LIN {X 0,Y 573.137,Z 463.185,A -85,B 0,C 180,E1 -2255.983,E2 -2255.983} C_VEL
LIN {X 0,Y 573.164,Z 455.803,A -85,B 0,C 180,E1 -2256.86,E2 -2256.86} C_VEL
LIN {X 0,Y 573.212,Z 448.405,A -85,B 0,C 180,E1 -2257.574,E2 -2257.574} C_VEL
LIN {X 0,Y 573.278,Z 440.543,A -85,B 0,C 180,E1 -2258.193,E2 -2258.193} C_VEL
LIN {X 0,Y 573.324,Z 430.729,A -85,B 0,C 180,E1 -2258.814,E2 -2258.814} C_VEL
LIN {X 0,Y 573.388,Z 419.304,A -85,B 0,C 180,E1 -2259.346,E2 -2259.346} C_VEL
LIN {X 0,Y 573.473,Z 409.247,A -85,B 0,C 180,E1 -2259.679,E2 -2259.679} C_VEL
LIN {X 0,Y 573.529,Z 400.443,A -85,B 0,C 180,E1 -2259.878,E2 -2259.878} C_VEL
LIN {X 0,Y 573.641,Z 328.384,A -85,B 0,C 180,E1 -2260.797,E2 -2260.797} C_VEL
LIN {X 0,Y 573.174,Z 322.224,A -85,B 0,C 180,E1 -2260.899,E2 -2260.899} C_VEL
LIN {X 0,Y 573.324,Z 304.046,A -85,B 0,C 180,E1 -2263.649,E2 -2263.649} C_VEL
LIN {X 0,Y 573.504,Z 285.12,A -85,B 0,C 180,E1 -2266.544,E2 -2266.544} C_VEL
LIN {X 0,Y 573.63,Z 266.907,A -85,B 0,C 180,E1 -2269.371,E2 -2269.371} C_VEL
LIN {X 0,Y 573.846,Z 250.306,A -85,B 0,C 180,E1 -2271.934,E2 -2271.934} C_VEL
LIN {X 0,Y 573.51,Z 245.432,A -85,B 0,C 180,E1 -2272.706,E2 -2272.706} C_VEL
LIN {X 0,Y 573.237,Z 243.895,A -85,B 0,C 180,E1 -2272.98,E2 -2272.98} C_VEL
LIN {X 0,Y 573.248,Z 243.895,A -85,B 0,C 180,E1 -2275.41,E2 -2275.41} C_VEL
LIN {X 0,Y 573.231,Z 243.888,A -85,B 0,C 180,E1 -2278.564,E2 -2278.564} C_VEL
LIN {X 0,Y 573.223,Z 243.891,A -85,B 0,C 180,E1 -2280.993,E2 -2280.993} C_VEL
LIN {X 0,Y 573.262,Z 243.894,A -85,B 0,C 180,E1 -2283.524,E2 -2283.524} C_VEL
LIN {X 0,Y 573.239,Z 243.889,A -85,B 0,C 180,E1 -2286.049,E2 -2286.049} C_VEL
LIN {X 0,Y 573.236,Z 243.887,A -85,B 0,C 180,E1 -2288.701,E2 -2288.701} C_VEL
LIN {X 0,Y 573.251,Z 243.894,A -85,B 0,C 180,E1 -2291.595,E2 -2291.595} C_VEL
LIN {X 0,Y 573.233,Z 243.887,A -85,B 0,C 180,E1 -2294.333,E2 -2294.333} C_VEL
LIN {X 0,Y 573.236,Z 243.894,A -85,B 0,C 180,E1 -2297.358,E2 -2297.358} C_VEL
LIN {X 0,Y 573.242,Z 243.886,A -85,B 0,C 180,E1 -2300.392,E2 -2300.392} C_VEL
LIN {X 0,Y 573.251,Z 243.888,A -85,B 0,C 180,E1 -2303.077,E2 -2303.077} C_VEL
LIN {X 0,Y 573.263,Z 243.891,A -85,B 0,C 180,E1 -2305.671,E2 -2305.671} C_VEL
LIN {X 0,Y 573.238,Z 243.888,A -85,B 0,C 180,E1 -2308.184,E2 -2308.184} C_VEL
LIN {X 0,Y 573.261,Z 243.884,A -85,B 0,C 180,E1 -2310.634,E2 -2310.634} C_VEL
LIN {X 0,Y 573.265,Z 243.893,A -85,B 0,C 180,E1 -2313.5,E2 -2313.5} C_VEL
LIN {X 0,Y 573.228,Z 243.889,A -85,B 0,C 180,E1 -2316.134,E2 -2316.134} C_VEL
LIN {X 0,Y 573.247,Z 243.89,A -85,B 0,C 180,E1 -2319.173,E2 -2319.173} C_VEL
LIN {X 0,Y 573.225,Z 243.896,A -85,B 0,C 180,E1 -2321.411,E2 -2321.411} C_VEL
LIN {X 0,Y 573.247,Z 243.894,A -85,B 0,C 180,E1 -2323.621,E2 -2323.621} C_VEL
LIN {X 0,Y 573.267,Z 243.889,A -85,B 0,C 180,E1 -2325.806,E2 -2325.806} C_VEL
LIN {X 0,Y 573.256,Z 243.885,A -85,B 0,C 180,E1 -2328.744,E2 -2328.744} C_VEL
LIN {X 0,Y 573.3,Z 243.889,A -85,B 0,C 180,E1 -2331.54,E2 -2331.54} C_VEL
LIN {X 0,Y 573.284,Z 243.881,A -85,B 0,C 180,E1 -2334.371,E2 -2334.371} C_VEL
LIN {X 0,Y 573.302,Z 243.883,A -85,B 0,C 180,E1 -2337.892,E2 -2337.892} C_VEL
LIN {X 0,Y 573.329,Z 243.875,A -85,B 0,C 180,E1 -2340.702,E2 -2340.702} C_VEL
LIN {X 0,Y 573.232,Z 243.897,A -85,B 0,C 180,E1 -2343.514,E2 -2343.514} C_VEL
LIN {X 0,Y 573.283,Z 243.89,A -85,B 0,C 180,E1 -2345.628,E2 -2345.628} C_VEL
LIN {X 0,Y 573.284,Z 243.881,A -85,B 0,C 180,E1 -2348.459,E2 -2348.459} C_VEL
LIN {X 0,Y 573.263,Z 243.89,A -85,B 0,C 180,E1 -2351.311,E2 -2351.311} C_VEL
LIN {X 0,Y 573.264,Z 243.885,A -85,B 0,C 180,E1 -2354.192,E2 -2354.192} C_VEL
LIN {X 0,Y 573.251,Z 243.888,A -85,B 0,C 180,E1 -2357.111,E2 -2357.111} C_VEL
LIN {X 0,Y 573.248,Z 243.888,A -85,B 0,C 180,E1 -2360.076,E2 -2360.076} C_VEL
LIN {X 0,Y 573.229,Z 243.888,A -85,B 0,C 180,E1 -2362.337,E2 -2362.337} C_VEL
LIN {X 0,Y 573.242,Z 243.886,A -85,B 0,C 180,E1 -2364.398,E2 -2364.398} C_VEL
LIN {X 0,Y 572.617,Z 243.967,A -85,B 0,C 180,E1 -2364.985,E2 -2364.985} C_VEL
LIN {X 0,Y 569.778,Z 244.324,A -85,B 0,C 180,E1 -2365.936,E2 -2365.936} C_VEL
LIN {X 0,Y 567.349,Z 244.629,A -85,B 0,C 180,E1 -2366.702,E2 -2366.702} C_VEL
LIN {X 0,Y 566.297,Z 244.758,A -85,B 0,C 180,E1 -2367.293,E2 -2367.293} C_VEL
LIN {X 0,Y 566.208,Z 244.767,A -85,B 0,C 180,E1 -2367.494,E2 -2367.494} C_VEL
LIN {X 0,Y 566.179,Z 244.766,A -85,B 0,C 180,E1 -2370.592,E2 -2370.592} C_VEL
LIN {X 0,Y 566.22,Z 244.764,A -85,B 0,C 180,E1 -2373.101,E2 -2373.101} C_VEL
LIN {X 0,Y 566.204,Z 244.771,A -85,B 0,C 180,E1 -2375.688,E2 -2375.688} C_VEL
LIN {X 0,Y 566.206,Z 244.763,A -85,B 0,C 180,E1 -2378.559,E2 -2378.559} C_VEL
LIN {X 0,Y 566.202,Z 244.767,A -85,B 0,C 180,E1 -2381.136,E2 -2381.136} C_VEL
LIN {X 0,Y 566.19,Z 244.768,A -85,B 0,C 180,E1 -2384.035,E2 -2384.035} C_VEL
LIN {X 0,Y 566.2,Z 244.766,A -85,B 0,C 180,E1 -2387.082,E2 -2387.082} C_VEL
LIN {X 0,Y 566.217,Z 244.767,A -85,B 0,C 180,E1 -2389.803,E2 -2389.803} C_VEL
LIN {X 0,Y 566.189,Z 244.765,A -85,B 0,C 180,E1 -2392.599,E2 -2392.599} C_VEL
LIN {X 0,Y 566.203,Z 244.767,A -85,B 0,C 180,E1 -2395.182,E2 -2395.182} C_VEL
LIN {X 0,Y 566.227,Z 244.767,A -85,B 0,C 180,E1 -2397.744,E2 -2397.744} C_VEL
LIN {X 0,Y 566.194,Z 244.765,A -85,B 0,C 180,E1 -2400.328,E2 -2400.328} C_VEL
LIN {X 0,Y 566.21,Z 244.762,A -85,B 0,C 180,E1 -2402.661,E2 -2402.661} C_VEL
LIN {X 0,Y 566.226,Z 244.763,A -85,B 0,C 180,E1 -2405.039,E2 -2405.039} C_VEL
LIN {X 0,Y 566.192,Z 244.771,A -85,B 0,C 180,E1 -2407.369,E2 -2407.369} C_VEL
LIN {X 0,Y 566.211,Z 244.771,A -85,B 0,C 180,E1 -2409.663,E2 -2409.663} C_VEL
LIN {X 0,Y 566.191,Z 244.765,A -85,B 0,C 180,E1 -2412.668,E2 -2412.668} C_VEL
LIN {X 0,Y 566.224,Z 244.77,A -85,B 0,C 180,E1 -2415.627,E2 -2415.627} C_VEL
LIN {X 0,Y 566.267,Z 244.755,A -85,B 0,C 180,E1 -2418.654,E2 -2418.654} C_VEL
LIN {X 0,Y 566.224,Z 244.768,A -85,B 0,C 180,E1 -2421.434,E2 -2421.434} C_VEL
LIN {X 0,Y 566.243,Z 244.759,A -85,B 0,C 180,E1 -2424.301,E2 -2424.301} C_VEL
LIN {X 0,Y 566.268,Z 244.759,A -85,B 0,C 180,E1 -2427.154,E2 -2427.154} C_VEL
LIN {X 0,Y 566.273,Z 244.758,A -85,B 0,C 180,E1 -2430,E2 -2430} C_VEL
LIN {X 0,Y 566.261,Z 244.757,A -85,B 0,C 180,E1 -2432.845,E2 -2432.845} C_VEL
LIN {X 0,Y 566.244,Z 244.766,A -85,B 0,C 180,E1 -2435.698,E2 -2435.698} C_VEL
LIN {X 0,Y 566.195,Z 244.764,A -85,B 0,C 180,E1 -2438.566,E2 -2438.566} C_VEL
LIN {X 0,Y 566.232,Z 244.768,A -85,B 0,C 180,E1 -2441.454,E2 -2441.454} C_VEL
LIN {X 0,Y 566.208,Z 244.763,A -85,B 0,C 180,E1 -2444.5,E2 -2444.5} C_VEL
LIN {X 0,Y 566.186,Z 244.771,A -85,B 0,C 180,E1 -2447.332,E2 -2447.332} C_VEL
LIN {X 0,Y 566.199,Z 244.764,A -85,B 0,C 180,E1 -2450.337,E2 -2450.337} C_VEL
LIN {X 0,Y 566.157,Z 244.774,A -85,B 0,C 180,E1 -2453.281,E2 -2453.281} C_VEL
LIN {X 0,Y 566.193,Z 244.772,A -85,B 0,C 180,E1 -2455.749,E2 -2455.749} C_VEL
LIN {X 0,Y 566.191,Z 244.766,A -85,B 0,C 180,E1 -2458.202,E2 -2458.202} C_VEL
LIN {X 0,Y 566.178,Z 244.769,A -85,B 0,C 180,E1 -2461.076,E2 -2461.076} C_VEL
LIN {X 0,Y 566.19,Z 244.872,A -85,B 0,C 180,E1 -2463.205,E2 -2463.205} C_VEL
LIN {X 0,Y 566.004,Z 257.339,A -85,B 0,C 180,E1 -2466.189,E2 -2466.189} C_VEL
LIN {X 0,Y 565.966,Z 265.195,A -85,B 0,C 180,E1 -2468.054,E2 -2468.054} C_VEL
LIN {X 0,Y 566.66,Z 271.612,A -85,B 0,C 180,E1 -2468.154,E2 -2468.154} C_VEL
LIN {X 0,Y 566.526,Z 339.502,A -85,B 0,C 180,E1 -2469.027,E2 -2469.027} C_VEL
LIN {X 0,Y 566.417,Z 349.053,A -85,B 0,C 180,E1 -2469.239,E2 -2469.239} C_VEL
LIN {X 0,Y 566.403,Z 358.967,A -85,B 0,C 180,E1 -2469.57,E2 -2469.57} C_VEL
LIN {X 0,Y 566.3,Z 369.307,A -85,B 0,C 180,E1 -2470.041,E2 -2470.041} C_VEL
LIN {X 0,Y 566.244,Z 379.006,A -85,B 0,C 180,E1 -2470.637,E2 -2470.637} C_VEL
LIN {X 0,Y 566.155,Z 387.059,A -85,B 0,C 180,E1 -2471.258,E2 -2471.258} C_VEL
LIN {X 0,Y 566.113,Z 394.356,A -85,B 0,C 180,E1 -2471.947,E2 -2471.947} C_VEL
LIN {X 0,Y 566.027,Z 400.004,A -85,B 0,C 180,E1 -2472.584,E2 -2472.584} C_VEL
LIN {X 0,Y 565.976,Z 405.227,A -85,B 0,C 180,E1 -2473.286,E2 -2473.286} C_VEL
LIN {X 0,Y 565.962,Z 409.981,A -85,B 0,C 180,E1 -2474.057,E2 -2474.057} C_VEL
LIN {X 0,Y 565.9,Z 414.867,A -85,B 0,C 180,E1 -2475.062,E2 -2475.062} C_VEL
LIN {X 0,Y 565.896,Z 418.093,A -85,B 0,C 180,E1 -2475.936,E2 -2475.936} C_VEL
LIN {X 0,Y 565.857,Z 421.152,A -85,B 0,C 180,E1 -2477.119,E2 -2477.119} C_VEL
LIN {X 0,Y 565.849,Z 422.627,A -85,B 0,C 180,E1 -2478.176,E2 -2478.176} C_VEL
LIN {X 0,Y 565.824,Z 422.932,A -85,B 0,C 180,E1 -2479.258,E2 -2479.258} C_VEL
LIN {X 0,Y 565.858,Z 422.084,A -85,B 0,C 180,E1 -2480.356,E2 -2480.356} C_VEL
LIN {X 0,Y 565.899,Z 419.695,A -85,B 0,C 180,E1 -2481.615,E2 -2481.615} C_VEL
LIN {X 0,Y 565.921,Z 416.514,A -85,B 0,C 180,E1 -2482.634,E2 -2482.634} C_VEL
LIN {X 0,Y 565.937,Z 412.077,A -85,B 0,C 180,E1 -2483.642,E2 -2483.642} C_VEL
LIN {X 0,Y 565.987,Z 407.261,A -85,B 0,C 180,E1 -2484.494,E2 -2484.494} C_VEL
LIN {X 0,Y 566.037,Z 402.656,A -85,B 0,C 180,E1 -2485.171,E2 -2485.171} C_VEL
LIN {X 0,Y 566.085,Z 395.37,A -85,B 0,C 180,E1 -2486.037,E2 -2486.037} C_VEL
LIN {X 0,Y 566.135,Z 388.686,A -85,B 0,C 180,E1 -2486.689,E2 -2486.689} C_VEL
LIN {X 0,Y 566.24,Z 381.192,A -85,B 0,C 180,E1 -2487.293,E2 -2487.293} C_VEL
LIN {X 0,Y 566.33,Z 374.361,A -85,B 0,C 180,E1 -2487.751,E2 -2487.751} C_VEL
LIN {X 0,Y 566.344,Z 365.709,A -85,B 0,C 180,E1 -2488.223,E2 -2488.223} C_VEL
LIN {X 0,Y 566.379,Z 357.089,A -85,B 0,C 180,E1 -2488.591,E2 -2488.591} C_VEL
LIN {X 0,Y 566.474,Z 347.518,A -85,B 0,C 180,E1 -2488.891,E2 -2488.891} C_VEL
LIN {X 0,Y 566.541,Z 337.573,A -85,B 0,C 180,E1 -2489.096,E2 -2489.096} C_VEL
LIN {X 0,Y 566.548,Z 269.023,A -85,B 0,C 180,E1 -2489.97,E2 -2489.97} C_VEL
LIN {X 0,Y 565.997,Z 265.17,A -85,B 0,C 180,E1 -2490.041,E2 -2490.041} C_VEL
LIN {X 0,Y 566.136,Z 252.55,A -85,B 0,C 180,E1 -2493.042,E2 -2493.042} C_VEL
LIN {X 0,Y 566.185,Z 244.77,A -85,B 0,C 180,E1 -2494.949,E2 -2494.949} C_VEL
LIN {X 0,Y 566.169,Z 244.769,A -85,B 0,C 180,E1 -2497.369,E2 -2497.369} C_VEL
LIN {X 0,Y 566.209,Z 244.764,A -85,B 0,C 180,E1 -2499.664,E2 -2499.664} C_VEL
LIN {X 0,Y 566.194,Z 244.772,A -85,B 0,C 180,E1 -2502.669,E2 -2502.669} C_VEL
LIN {X 0,Y 566.222,Z 244.761,A -85,B 0,C 180,E1 -2505.627,E2 -2505.627} C_VEL
LIN {X 0,Y 566.264,Z 244.763,A -85,B 0,C 180,E1 -2508.655,E2 -2508.655} C_VEL
LIN {X 0,Y 566.239,Z 244.759,A -85,B 0,C 180,E1 -2511.435,E2 -2511.435} C_VEL
LIN {X 0,Y 566.251,Z 244.764,A -85,B 0,C 180,E1 -2514.302,E2 -2514.302} C_VEL
LIN {X 0,Y 566.271,Z 244.755,A -85,B 0,C 180,E1 -2517.867,E2 -2517.867} C_VEL
LIN {X 0,Y 566.298,Z 244.757,A -85,B 0,C 180,E1 -2520.712,E2 -2520.712} C_VEL
LIN {X 0,Y 566.27,Z 244.759,A -85,B 0,C 180,E1 -2522.846,E2 -2522.846} C_VEL
LIN {X 0,Y 566.252,Z 244.757,A -85,B 0,C 180,E1 -2525.699,E2 -2525.699} C_VEL
LIN {X 0,Y 566.239,Z 244.768,A -85,B 0,C 180,E1 -2528.566,E2 -2528.566} C_VEL
LIN {X 0,Y 566.232,Z 244.759,A -85,B 0,C 180,E1 -2531.455,E2 -2531.455} C_VEL
LIN {X 0,Y 566.225,Z 244.77,A -85,B 0,C 180,E1 -2534.507,E2 -2534.507} C_VEL
LIN {X 0,Y 566.196,Z 244.763,A -85,B 0,C 180,E1 -2537.332,E2 -2537.332} C_VEL
LIN {X 0,Y 566.212,Z 244.769,A -85,B 0,C 180,E1 -2540.338,E2 -2540.338} C_VEL
LIN {X 0,Y 566.182,Z 244.765,A -85,B 0,C 180,E1 -2543.405,E2 -2543.405} C_VEL
LIN {X 0,Y 566.219,Z 244.76,A -85,B 0,C 180,E1 -2545.749,E2 -2545.749} C_VEL
LIN {X 0,Y 566.201,Z 244.769,A -85,B 0,C 180,E1 -2548.204,E2 -2548.204} C_VEL
LIN {X 0,Y 566.181,Z 244.774,A -85,B 0,C 180,E1 -2550.593,E2 -2550.593} C_VEL
LIN {X 0,Y 566.223,Z 244.761,A -85,B 0,C 180,E1 -2553.102,E2 -2553.102} C_VEL
LIN {X 0,Y 566.206,Z 244.763,A -85,B 0,C 180,E1 -2555.689,E2 -2555.689} C_VEL
LIN {X 0,Y 566.209,Z 244.772,A -85,B 0,C 180,E1 -2558.56,E2 -2558.56} C_VEL
LIN {X 0,Y 566.203,Z 244.764,A -85,B 0,C 180,E1 -2561.137,E2 -2561.137} C_VEL
LIN {X 0,Y 566.192,Z 244.767,A -85,B 0,C 180,E1 -2564.037,E2 -2564.037} C_VEL
LIN {X 0,Y 566.197,Z 244.766,A -85,B 0,C 180,E1 -2567.084,E2 -2567.084} C_VEL
LIN {X 0,Y 566.203,Z 244.764,A -85,B 0,C 180,E1 -2569.802,E2 -2569.802} C_VEL
LIN {X 0,Y 566.195,Z 244.773,A -85,B 0,C 180,E1 -2572.6,E2 -2572.6} C_VEL
LIN {X 0,Y 566.204,Z 244.764,A -85,B 0,C 180,E1 -2575.183,E2 -2575.183} C_VEL
LIN {X 0,Y 566.227,Z 244.761,A -85,B 0,C 180,E1 -2577.744,E2 -2577.744} C_VEL
LIN {X 0,Y 566.2,Z 244.772,A -85,B 0,C 180,E1 -2580.329,E2 -2580.329} C_VEL
LIN {X 0,Y 566.195,Z 244.765,A -85,B 0,C 180,E1 -2583.344,E2 -2583.344} C_VEL
LIN {X 0,Y 566.198,Z 244.767,A -85,B 0,C 180,E1 -2585.82,E2 -2585.82} C_VEL
LIN {X 0,Y 566.223,Z 244.825,A -85,B 0,C 180,E1 -2587.049,E2 -2587.049} C_VEL
LIN {X 0,Y 566.789,Z 249.5,A -85,B 0,C 180,E1 -2587.779,E2 -2587.779} C_VEL
LIN {X 0,Y 566.638,Z 267.218,A -85,B 0,C 180,E1 -2590.498,E2 -2590.498} C_VEL
LIN {X 0,Y 566.491,Z 286.246,A -85,B 0,C 180,E1 -2593.421,E2 -2593.421} C_VEL
LIN {X 0,Y 566.283,Z 305.235,A -85,B 0,C 180,E1 -2596.361,E2 -2596.361} C_VEL
LIN {X 0,Y 566.128,Z 322.265,A -85,B 0,C 180,E1 -2598.97,E2 -2598.97} C_VEL
LIN {X 0,Y 566.696,Z 329.655,A -85,B 0,C 180,E1 -2599.085,E2 -2599.085} C_VEL
LIN {X 0,Y 566.59,Z 399.161,A -85,B 0,C 180,E1 -2599.977,E2 -2599.977} C_VEL
LIN {X 0,Y 566.469,Z 408.425,A -85,B 0,C 180,E1 -2600.178,E2 -2600.178} C_VEL
LIN {X 0,Y 566.425,Z 416.897,A -85,B 0,C 180,E1 -2600.448,E2 -2600.448} C_VEL
LIN {X 0,Y 566.358,Z 425.402,A -85,B 0,C 180,E1 -2600.807,E2 -2600.807} C_VEL
LIN {X 0,Y 566.318,Z 433.733,A -85,B 0,C 180,E1 -2601.256,E2 -2601.256} C_VEL
LIN {X 0,Y 566.212,Z 441.771,A -85,B 0,C 180,E1 -2601.794,E2 -2601.794} C_VEL
LIN {X 0,Y 566.12,Z 450.435,A -85,B 0,C 180,E1 -2602.51,E2 -2602.51} C_VEL
LIN {X 0,Y 566.088,Z 458.908,A -85,B 0,C 180,E1 -2603.402,E2 -2603.402} C_VEL
LIN {X 0,Y 566.057,Z 464.437,A -85,B 0,C 180,E1 -2604.121,E2 -2604.121} C_VEL
LIN {X 0,Y 565.906,Z 469.99,A -85,B 0,C 180,E1 -2605.013,E2 -2605.013} C_VEL
LIN {X 0,Y 565.944,Z 475.15,A -85,B 0,C 180,E1 -2606.084,E2 -2606.084} C_VEL
LIN {X 0,Y 565.88,Z 478.936,A -85,B 0,C 180,E1 -2607.153,E2 -2607.153} C_VEL
LIN {X 0,Y 565.841,Z 480.683,A -85,B 0,C 180,E1 -2607.865,E2 -2607.865} C_VEL
LIN {X 0,Y 565.844,Z 481.933,A -85,B 0,C 180,E1 -2608.577,E2 -2608.577} C_VEL
LIN {X 0,Y 565.837,Z 482.709,A -85,B 0,C 180,E1 -2609.289,E2 -2609.289} C_VEL
LIN {X 0,Y 565.836,Z 483,A -85,B 0,C 180,E1 -2610,E2 -2610} C_VEL
LIN {X 0,Y 565.837,Z 482.708,A -85,B 0,C 180,E1 -2610.712,E2 -2610.712} C_VEL
LIN {X 0,Y 565.844,Z 481.932,A -85,B 0,C 180,E1 -2611.424,E2 -2611.424} C_VEL
LIN {X 0,Y 565.841,Z 480.681,A -85,B 0,C 180,E1 -2612.136,E2 -2612.136} C_VEL
LIN {X 0,Y 565.912,Z 477.787,A -85,B 0,C 180,E1 -2613.204,E2 -2613.204} C_VEL
LIN {X 0,Y 565.944,Z 475.148,A -85,B 0,C 180,E1 -2613.916,E2 -2613.916} C_VEL
LIN {X 0,Y 565.906,Z 469.985,A -85,B 0,C 180,E1 -2614.987,E2 -2614.987} C_VEL
LIN {X 0,Y 566.082,Z 463.184,A -85,B 0,C 180,E1 -2616.058,E2 -2616.058} C_VEL
LIN {X 0,Y 566.092,Z 456.178,A -85,B 0,C 180,E1 -2616.906,E2 -2616.906} C_VEL
LIN {X 0,Y 566.146,Z 448.403,A -85,B 0,C 180,E1 -2617.669,E2 -2617.669} C_VEL
LIN {X 0,Y 566.258,Z 440.54,A -85,B 0,C 180,E1 -2618.296,E2 -2618.296} C_VEL
LIN {X 0,Y 566.327,Z 432.227,A -85,B 0,C 180,E1 -2618.834,E2 -2618.834} C_VEL
LIN {X 0,Y 566.374,Z 421.612,A -85,B 0,C 180,E1 -2619.373,E2 -2619.373} C_VEL
LIN {X 0,Y 566.473,Z 410.078,A -85,B 0,C 180,E1 -2619.777,E2 -2619.777} C_VEL
LIN {X 0,Y 566.559,Z 400.442,A -85,B 0,C 180,E1 -2620.001,E2 -2620.001} C_VEL
LIN {X 0,Y 566.686,Z 331.981,A -85,B 0,C 180,E1 -2620.885,E2 -2620.885} C_VEL
LIN {X 0,Y 566.411,Z 324.693,A -85,B 0,C 180,E1 -2620.983,E2 -2620.983} C_VEL
LIN {X 0,Y 566.137,Z 322.13,A -85,B 0,C 180,E1 -2621.051,E2 -2621.051} C_VEL
LIN {X 0,Y 566.319,Z 304.046,A -85,B 0,C 180,E1 -2623.821,E2 -2623.821} C_VEL
LIN {X 0,Y 566.512,Z 284.258,A -85,B 0,C 180,E1 -2626.889,E2 -2626.889} C_VEL
LIN {X 0,Y 566.634,Z 266.984,A -85,B 0,C 180,E1 -2629.565,E2 -2629.565} C_VEL
LIN {X 0,Y 566.902,Z 250.013,A -85,B 0,C 180,E1 -2632.217,E2 -2632.217} C_VEL
LIN {X 0,Y 566.191,Z 244.774,A -85,B 0,C 180,E1 -2633.099,E2 -2633.099} C_VEL
LIN {X 0,Y 566.207,Z 244.77,A -85,B 0,C 180,E1 -2635.749,E2 -2635.749} C_VEL
LIN {X 0,Y 566.203,Z 244.764,A -85,B 0,C 180,E1 -2638.202,E2 -2638.202} C_VEL
LIN {X 0,Y 566.189,Z 244.768,A -85,B 0,C 180,E1 -2641.076,E2 -2641.076} C_VEL
LIN {X 0,Y 566.211,Z 244.768,A -85,B 0,C 180,E1 -2643.734,E2 -2643.734} C_VEL
LIN {X 0,Y 566.207,Z 244.762,A -85,B 0,C 180,E1 -2646.569,E2 -2646.569} C_VEL
LIN {X 0,Y 566.212,Z 244.769,A -85,B 0,C 180,E1 -2649.685,E2 -2649.685} C_VEL
LIN {X 0,Y 566.211,Z 244.764,A -85,B 0,C 180,E1 -2652.087,E2 -2652.087} C_VEL
LIN {X 0,Y 566.171,Z 244.77,A -85,B 0,C 180,E1 -2655.035,E2 -2655.035} C_VEL
LIN {X 0,Y 566.209,Z 244.764,A -85,B 0,C 180,E1 -2658.136,E2 -2658.136} C_VEL
LIN {X 0,Y 566.216,Z 244.762,A -85,B 0,C 180,E1 -2660.726,E2 -2660.726} C_VEL
LIN {X 0,Y 566.203,Z 244.769,A -85,B 0,C 180,E1 -2663.784,E2 -2663.784} C_VEL
LIN {X 0,Y 566.207,Z 244.763,A -85,B 0,C 180,E1 -2666.265,E2 -2666.265} C_VEL
LIN {X 0,Y 566.186,Z 244.767,A -85,B 0,C 180,E1 -2668.923,E2 -2668.923} C_VEL
LIN {X 0,Y 566.224,Z 244.765,A -85,B 0,C 180,E1 -2671.858,E2 -2671.858} C_VEL
LIN {X 0,Y 566.221,Z 244.761,A -85,B 0,C 180,E1 -2674.251,E2 -2674.251} C_VEL
LIN {X 0,Y 566.186,Z 244.765,A -85,B 0,C 180,E1 -2676.713,E2 -2676.713} C_VEL
LIN {X 0,Y 566.21,Z 244.77,A -85,B 0,C 180,E1 -2679.662,E2 -2679.662} C_VEL
LIN {X 0,Y 566.194,Z 244.764,A -85,B 0,C 180,E1 -2682.668,E2 -2682.668} C_VEL
LIN {X 0,Y 566.228,Z 244.769,A -85,B 0,C 180,E1 -2685.626,E2 -2685.626} C_VEL
LIN {X 0,Y 566.228,Z 244.76,A -85,B 0,C 180,E1 -2688.674,E2 -2688.674} C_VEL
LIN {X 0,Y 566.241,Z 244.767,A -85,B 0,C 180,E1 -2691.434,E2 -2691.434} C_VEL
LIN {X 0,Y 566.253,Z 244.757,A -85,B 0,C 180,E1 -2694.301,E2 -2694.301} C_VEL
LIN {X 0,Y 566.274,Z 244.759,A -85,B 0,C 180,E1 -2697.866,E2 -2697.866} C_VEL
LIN {X 0,Y 566.299,Z 244.751,A -85,B 0,C 180,E1 -2700.71,E2 -2700.71} C_VEL
LIN {X 0,Y 566.271,Z 244.755,A -85,B 0,C 180,E1 -2702.845,E2 -2702.845} C_VEL
LIN {X 0,Y 566.251,Z 244.765,A -85,B 0,C 180,E1 -2705.698,E2 -2705.698} C_VEL
LIN {X 0,Y 566.228,Z 244.76,A -85,B 0,C 180,E1 -2708.565,E2 -2708.565} C_VEL
LIN {X 0,Y 566.233,Z 244.768,A -85,B 0,C 180,E1 -2711.454,E2 -2711.454} C_VEL
LIN {X 0,Y 566.225,Z 244.76,A -85,B 0,C 180,E1 -2714.506,E2 -2714.506} C_VEL
LIN {X 0,Y 566.196,Z 244.77,A -85,B 0,C 180,E1 -2717.331,E2 -2717.331} C_VEL
LIN {X 0,Y 566.211,Z 244.762,A -85,B 0,C 180,E1 -2720.336,E2 -2720.336} C_VEL
LIN {X 0,Y 566.18,Z 244.773,A -85,B 0,C 180,E1 -2723.403,E2 -2723.403} C_VEL
LIN {X 0,Y 566.217,Z 244.768,A -85,B 0,C 180,E1 -2725.748,E2 -2725.748} C_VEL
LIN {X 0,Y 566.208,Z 244.767,A -85,B 0,C 180,E1 -2727.494,E2 -2727.494} C_VEL
LIN {X 0,Y 565.528,Z 244.85,A -85,B 0,C 180,E1 -2728.087,E2 -2728.087} C_VEL
LIN {X 0,Y 562.657,Z 245.207,A -85,B 0,C 180,E1 -2729.051,E2 -2729.051} C_VEL
LIN {X 0,Y 560.243,Z 245.511,A -85,B 0,C 180,E1 -2729.826,E2 -2729.826} C_VEL
LIN {X 0,Y 559.215,Z 245.634,A -85,B 0,C 180,E1 -2730.425,E2 -2730.425} C_VEL
LIN {X 0,Y 559.136,Z 245.643,A -85,B 0,C 180,E1 -2730.628,E2 -2730.628} C_VEL
LIN {X 0,Y 559.169,Z 245.649,A -85,B 0,C 180,E1 -2733.573,E2 -2733.573} C_VEL
LIN {X 0,Y 559.16,Z 245.641,A -85,B 0,C 180,E1 -2736.448,E2 -2736.448} C_VEL
LIN {X 0,Y 559.168,Z 245.641,A -85,B 0,C 180,E1 -2738.933,E2 -2738.933} C_VEL
LIN {X 0,Y 559.182,Z 245.644,A -85,B 0,C 180,E1 -2741.767,E2 -2741.767} C_VEL
LIN {X 0,Y 559.13,Z 245.645,A -85,B 0,C 180,E1 -2744.739,E2 -2744.739} C_VEL
LIN {X 0,Y 559.158,Z 245.646,A -85,B 0,C 180,E1 -2747.257,E2 -2747.257} C_VEL
LIN {X 0,Y 559.176,Z 245.64,A -85,B 0,C 180,E1 -2750.135,E2 -2750.135} C_VEL
LIN {X 0,Y 559.134,Z 245.645,A -85,B 0,C 180,E1 -2752.892,E2 -2752.892} C_VEL
LIN {X 0,Y 559.157,Z 245.644,A -85,B 0,C 180,E1 -2756.05,E2 -2756.05} C_VEL
LIN {X 0,Y 559.154,Z 245.643,A -85,B 0,C 180,E1 -2758.981,E2 -2758.981} C_VEL
LIN {X 0,Y 559.183,Z 245.638,A -85,B 0,C 180,E1 -2762.288,E2 -2762.288} C_VEL
LIN {X 0,Y 559.169,Z 245.64,A -85,B 0,C 180,E1 -2764.813,E2 -2764.813} C_VEL
LIN {X 0,Y 559.153,Z 245.644,A -85,B 0,C 180,E1 -2767.068,E2 -2767.068} C_VEL
LIN {X 0,Y 559.177,Z 245.645,A -85,B 0,C 180,E1 -2769.396,E2 -2769.396} C_VEL
LIN {X 0,Y 559.139,Z 245.651,A -85,B 0,C 180,E1 -2771.686,E2 -2771.686} C_VEL
LIN {X 0,Y 559.161,Z 245.644,A -85,B 0,C 180,E1 -2773.948,E2 -2773.948} C_VEL
LIN {X 0,Y 559.163,Z 245.642,A -85,B 0,C 180,E1 -2776.184,E2 -2776.184} C_VEL
LIN {X 0,Y 559.201,Z 245.639,A -85,B 0,C 180,E1 -2779.134,E2 -2779.134} C_VEL
LIN {X 0,Y 559.196,Z 245.639,A -85,B 0,C 180,E1 -2782.053,E2 -2782.053} C_VEL
LIN {X 0,Y 559.246,Z 245.631,A -85,B 0,C 180,E1 -2784.953,E2 -2784.953} C_VEL
LIN {X 0,Y 559.236,Z 245.637,A -85,B 0,C 180,E1 -2787.839,E2 -2787.839} C_VEL
LIN {X 0,Y 559.26,Z 245.628,A -85,B 0,C 180,E1 -2790.72,E2 -2790.72} C_VEL
LIN {X 0,Y 559.228,Z 245.633,A -85,B 0,C 180,E1 -2792.881,E2 -2792.881} C_VEL
LIN {X 0,Y 559.211,Z 245.641,A -85,B 0,C 180,E1 -2795.77,E2 -2795.77} C_VEL
LIN {X 0,Y 559.16,Z 245.641,A -85,B 0,C 180,E1 -2798.674,E2 -2798.674} C_VEL
LIN {X 0,Y 559.195,Z 245.646,A -85,B 0,C 180,E1 -2801.6,E2 -2801.6} C_VEL
LIN {X 0,Y 559.169,Z 245.639,A -85,B 0,C 180,E1 -2804.587,E2 -2804.587} C_VEL
LIN {X 0,Y 559.145,Z 245.652,A -85,B 0,C 180,E1 -2807.557,E2 -2807.557} C_VEL
LIN {X 0,Y 559.157,Z 245.647,A -85,B 0,C 180,E1 -2809.837,E2 -2809.837} C_VEL
LIN {X 0,Y 559.128,Z 245.647,A -85,B 0,C 180,E1 -2812.153,E2 -2812.153} C_VEL
LIN {X 0,Y 559.136,Z 245.649,A -85,B 0,C 180,E1 -2815.299,E2 -2815.299} C_VEL
LIN {X 0,Y 559.13,Z 245.652,A -85,B 0,C 180,E1 -2817.714,E2 -2817.714} C_VEL
LIN {X 0,Y 559.138,Z 245.645,A -85,B 0,C 180,E1 -2820.183,E2 -2820.183} C_VEL
LIN {X 0,Y 559.146,Z 245.647,A -85,B 0,C 180,E1 -2823.144,E2 -2823.144} C_VEL
LIN {X 0,Y 559.081,Z 246.203,A -85,B 0,C 180,E1 -2823.364,E2 -2823.364} C_VEL
LIN {X 0,Y 558.961,Z 258.174,A -85,B 0,C 180,E1 -2826.223,E2 -2826.223} C_VEL
LIN {X 0,Y 558.906,Z 265.204,A -85,B 0,C 180,E1 -2827.916,E2 -2827.916} C_VEL
LIN {X 0,Y 559.692,Z 271.401,A -85,B 0,C 180,E1 -2828.015,E2 -2828.015} C_VEL
LIN {X 0,Y 559.549,Z 340.384,A -85,B 0,C 180,E1 -2828.916,E2 -2828.916} C_VEL
LIN {X 0,Y 559.438,Z 350.568,A -85,B 0,C 180,E1 -2829.157,E2 -2829.157} C_VEL
LIN {X 0,Y 559.348,Z 361.714,A -85,B 0,C 180,E1 -2829.558,E2 -2829.558} C_VEL
LIN {X 0,Y 559.265,Z 372.601,A -85,B 0,C 180,E1 -2830.122,E2 -2830.122} C_VEL
LIN {X 0,Y 559.194,Z 381.214,A -85,B 0,C 180,E1 -2830.694,E2 -2830.694} C_VEL
LIN {X 0,Y 559.093,Z 389.596,A -85,B 0,C 180,E1 -2831.385,E2 -2831.385} C_VEL
LIN {X 0,Y 558.975,Z 397.888,A -85,B 0,C 180,E1 -2832.236,E2 -2832.236} C_VEL
LIN {X 0,Y 558.912,Z 404.963,A -85,B 0,C 180,E1 -2833.172,E2 -2833.172} C_VEL
LIN {X 0,Y 558.867,Z 409.934,A -85,B 0,C 180,E1 -2833.985,E2 -2833.985} C_VEL
LIN {X 0,Y 558.846,Z 413.842,A -85,B 0,C 180,E1 -2834.768,E2 -2834.768} C_VEL
LIN {X 0,Y 558.81,Z 417.77,A -85,B 0,C 180,E1 -2835.795,E2 -2835.795} C_VEL
LIN {X 0,Y 558.799,Z 419.162,A -85,B 0,C 180,E1 -2836.234,E2 -2836.234} C_VEL
LIN {X 0,Y 558.753,Z 421.398,A -85,B 0,C 180,E1 -2837.219,E2 -2837.219} C_VEL
LIN {X 0,Y 558.753,Z 422.645,A -85,B 0,C 180,E1 -2838.194,E2 -2838.194} C_VEL
LIN {X 0,Y 558.741,Z 422.978,A -85,B 0,C 180,E1 -2839.152,E2 -2839.152} C_VEL
LIN {X 0,Y 558.752,Z 422.434,A -85,B 0,C 180,E1 -2840.107,E2 -2840.107} C_VEL
LIN {X 0,Y 558.758,Z 420.602,A -85,B 0,C 180,E1 -2841.243,E2 -2841.243} C_VEL
LIN {X 0,Y 558.818,Z 417.43,A -85,B 0,C 180,E1 -2842.401,E2 -2842.401} C_VEL
LIN {X 0,Y 558.845,Z 412.629,A -85,B 0,C 180,E1 -2843.595,E2 -2843.595} C_VEL
LIN {X 0,Y 558.912,Z 406.627,A -85,B 0,C 180,E1 -2844.661,E2 -2844.661} C_VEL
LIN {X 0,Y 558.95,Z 402.07,A -85,B 0,C 180,E1 -2845.324,E2 -2845.324} C_VEL
LIN {X 0,Y 559.014,Z 395.87,A -85,B 0,C 180,E1 -2846.072,E2 -2846.072} C_VEL
LIN {X 0,Y 559.091,Z 389.138,A -85,B 0,C 180,E1 -2846.745,E2 -2846.745} C_VEL
LIN {X 0,Y 559.214,Z 380.916,A -85,B 0,C 180,E1 -2847.418,E2 -2847.418} C_VEL
LIN {X 0,Y 559.321,Z 373.119,A -85,B 0,C 180,E1 -2847.936,E2 -2847.936} C_VEL
LIN {X 0,Y 559.34,Z 365.039,A -85,B 0,C 180,E1 -2848.372,E2 -2848.372} C_VEL
LIN {X 0,Y 559.429,Z 355.925,A -85,B 0,C 180,E1 -2848.754,E2 -2848.754} C_VEL
LIN {X 0,Y 559.49,Z 344.628,A -85,B 0,C 180,E1 -2849.094,E2 -2849.094} C_VEL
LIN {X 0,Y 559.544,Z 329.664,A -85,B 0,C 180,E1 -2849.333,E2 -2849.333} C_VEL
LIN {X 0,Y 559.654,Z 270.209,A -85,B 0,C 180,E1 -2850.091,E2 -2850.091} C_VEL
LIN {X 0,Y 558.935,Z 265.184,A -85,B 0,C 180,E1 -2850.178,E2 -2850.178} C_VEL
LIN {X 0,Y 559.056,Z 252.919,A -85,B 0,C 180,E1 -2853.093,E2 -2853.093} C_VEL
LIN {X 0,Y 559.096,Z 245.657,A -85,B 0,C 180,E1 -2854.699,E2 -2854.699} C_VEL
LIN {X 0,Y 559.111,Z 245.65,A -85,B 0,C 180,E1 -2857.067,E2 -2857.067} C_VEL
LIN {X 0,Y 559.175,Z 245.641,A -85,B 0,C 180,E1 -2859.396,E2 -2859.396} C_VEL
LIN {X 0,Y 559.145,Z 245.644,A -85,B 0,C 180,E1 -2861.687,E2 -2861.687} C_VEL
LIN {X 0,Y 559.161,Z 245.643,A -85,B 0,C 180,E1 -2863.949,E2 -2863.949} C_VEL
LIN {X 0,Y 559.163,Z 245.645,A -85,B 0,C 180,E1 -2866.185,E2 -2866.185} C_VEL
LIN {X 0,Y 559.2,Z 245.637,A -85,B 0,C 180,E1 -2869.134,E2 -2869.134} C_VEL
LIN {X 0,Y 559.2,Z 245.639,A -85,B 0,C 180,E1 -2872.054,E2 -2872.054} C_VEL
LIN {X 0,Y 559.251,Z 245.632,A -85,B 0,C 180,E1 -2874.954,E2 -2874.954} C_VEL
LIN {X 0,Y 559.243,Z 245.631,A -85,B 0,C 180,E1 -2877.84,E2 -2877.84} C_VEL
LIN {X 0,Y 559.268,Z 245.633,A -85,B 0,C 180,E1 -2880.721,E2 -2880.721} C_VEL
LIN {X 0,Y 559.236,Z 245.635,A -85,B 0,C 180,E1 -2882.882,E2 -2882.882} C_VEL
LIN {X 0,Y 559.221,Z 245.633,A -85,B 0,C 180,E1 -2885.771,E2 -2885.771} C_VEL
LIN {X 0,Y 559.194,Z 245.643,A -85,B 0,C 180,E1 -2888.675,E2 -2888.675} C_VEL
LIN {X 0,Y 559.196,Z 245.636,A -85,B 0,C 180,E1 -2891.601,E2 -2891.601} C_VEL
LIN {X 0,Y 559.19,Z 245.645,A -85,B 0,C 180,E1 -2894.596,E2 -2894.596} C_VEL
LIN {X 0,Y 559.155,Z 245.64,A -85,B 0,C 180,E1 -2897.557,E2 -2897.557} C_VEL
LIN {X 0,Y 559.167,Z 245.64,A -85,B 0,C 180,E1 -2899.838,E2 -2899.838} C_VEL
LIN {X 0,Y 559.135,Z 245.647,A -85,B 0,C 180,E1 -2902.153,E2 -2902.153} C_VEL
LIN {X 0,Y 559.172,Z 245.638,A -85,B 0,C 180,E1 -2905.188,E2 -2905.188} C_VEL
LIN {X 0,Y 559.188,Z 245.637,A -85,B 0,C 180,E1 -2907.712,E2 -2907.712} C_VEL
LIN {X 0,Y 559.159,Z 245.644,A -85,B 0,C 180,E1 -2910.183,E2 -2910.183} C_VEL
LIN {X 0,Y 559.169,Z 245.644,A -85,B 0,C 180,E1 -2912.715,E2 -2912.715} C_VEL
LIN {X 0,Y 559.151,Z 245.642,A -85,B 0,C 180,E1 -2915.323,E2 -2915.323} C_VEL
LIN {X 0,Y 559.129,Z 245.646,A -85,B 0,C 180,E1 -2918.018,E2 -2918.018} C_VEL
LIN {X 0,Y 559.17,Z 245.644,A -85,B 0,C 180,E1 -2920.811,E2 -2920.811} C_VEL
LIN {X 0,Y 559.136,Z 245.644,A -85,B 0,C 180,E1 -2923.735,E2 -2923.735} C_VEL
LIN {X 0,Y 559.141,Z 245.648,A -85,B 0,C 180,E1 -2926.804,E2 -2926.804} C_VEL
LIN {X 0,Y 559.155,Z 245.642,A -85,B 0,C 180,E1 -2929.189,E2 -2929.189} C_VEL
LIN {X 0,Y 559.129,Z 245.647,A -85,B 0,C 180,E1 -2931.983,E2 -2931.983} C_VEL
LIN {X 0,Y 559.143,Z 245.648,A -85,B 0,C 180,E1 -2934.786,E2 -2934.786} C_VEL
LIN {X 0,Y 559.171,Z 245.64,A -85,B 0,C 180,E1 -2937.362,E2 -2937.362} C_VEL
LIN {X 0,Y 559.145,Z 245.648,A -85,B 0,C 180,E1 -2940.144,E2 -2940.144} C_VEL
LIN {X 0,Y 559.163,Z 245.642,A -85,B 0,C 180,E1 -2943.175,E2 -2943.175} C_VEL
LIN {X 0,Y 559.156,Z 245.643,A -85,B 0,C 180,E1 -2945.496,E2 -2945.496} C_VEL
LIN {X 0,Y 559.202,Z 245.837,A -85,B 0,C 180,E1 -2946.998,E2 -2946.998} C_VEL
LIN {X 0,Y 559.777,Z 251.397,A -85,B 0,C 180,E1 -2947.874,E2 -2947.874} C_VEL
LIN {X 0,Y 559.602,Z 267.581,A -85,B 0,C 180,E1 -2950.377,E2 -2950.377} C_VEL
LIN {X 0,Y 559.477,Z 284.254,A -85,B 0,C 180,E1 -2952.952,E2 -2952.952} C_VEL
LIN {X 0,Y 559.318,Z 304.048,A -85,B 0,C 180,E1 -2956.003,E2 -2956.003} C_VEL
LIN {X 0,Y 559.09,Z 322.26,A -85,B 0,C 180,E1 -2958.828,E2 -2958.828} C_VEL
LIN {X 0,Y 559.72,Z 329.246,A -85,B 0,C 180,E1 -2958.942,E2 -2958.942} C_VEL
LIN {X 0,Y 559.611,Z 399.161,A -85,B 0,C 180,E1 -2959.851,E2 -2959.851} C_VEL
LIN {X 0,Y 559.494,Z 408.425,A -85,B 0,C 180,E1 -2960.054,E2 -2960.054} C_VEL
LIN {X 0,Y 559.441,Z 416.895,A -85,B 0,C 180,E1 -2960.327,E2 -2960.327} C_VEL
LIN {X 0,Y 559.363,Z 425.399,A -85,B 0,C 180,E1 -2960.691,E2 -2960.691} C_VEL
LIN {X 0,Y 559.308,Z 433.73,A -85,B 0,C 180,E1 -2961.146,E2 -2961.146} C_VEL
LIN {X 0,Y 559.198,Z 441.768,A -85,B 0,C 180,E1 -2961.69,E2 -2961.69} C_VEL
LIN {X 0,Y 559.094,Z 450.436,A -85,B 0,C 180,E1 -2962.416,E2 -2962.416} C_VEL
LIN {X 0,Y 559.034,Z 458.737,A -85,B 0,C 180,E1 -2963.297,E2 -2963.297} C_VEL
LIN {X 0,Y 559.004,Z 464.438,A -85,B 0,C 180,E1 -2964.047,E2 -2964.047} C_VEL
LIN {X 0,Y 558.822,Z 469.99,A -85,B 0,C 180,E1 -2964.95,E2 -2964.95} C_VEL
LIN {X 0,Y 558.859,Z 475.15,A -85,B 0,C 180,E1 -2966.034,E2 -2966.034} C_VEL
LIN {X 0,Y 558.803,Z 478.937,A -85,B 0,C 180,E1 -2967.117,E2 -2967.117} C_VEL
LIN {X 0,Y 558.747,Z 480.683,A -85,B 0,C 180,E1 -2967.838,E2 -2967.838} C_VEL
LIN {X 0,Y 558.744,Z 481.932,A -85,B 0,C 180,E1 -2968.559,E2 -2968.559} C_VEL
LIN {X 0,Y 558.737,Z 482.708,A -85,B 0,C 180,E1 -2969.279,E2 -2969.279} C_VEL
LIN {X 0,Y 558.737,Z 483,A -85,B 0,C 180,E1 -2970,E2 -2970} C_VEL
LIN {X 0,Y 558.737,Z 482.708,A -85,B 0,C 180,E1 -2970.721,E2 -2970.721} C_VEL
LIN {X 0,Y 558.744,Z 481.931,A -85,B 0,C 180,E1 -2971.442,E2 -2971.442} C_VEL
LIN {X 0,Y 558.747,Z 480.681,A -85,B 0,C 180,E1 -2972.163,E2 -2972.163} C_VEL
LIN {X 0,Y 558.836,Z 477.786,A -85,B 0,C 180,E1 -2973.244,E2 -2973.244} C_VEL
LIN {X 0,Y 558.859,Z 475.148,A -85,B 0,C 180,E1 -2973.966,E2 -2973.966} C_VEL
LIN {X 0,Y 558.822,Z 469.986,A -85,B 0,C 180,E1 -2975.051,E2 -2975.051} C_VEL
LIN {X 0,Y 559.018,Z 463.183,A -85,B 0,C 180,E1 -2976.135,E2 -2976.135} C_VEL
LIN {X 0,Y 559.036,Z 455.742,A -85,B 0,C 180,E1 -2977.04,E2 -2977.04} C_VEL
LIN {X 0,Y 559.119,Z 448.4,A -85,B 0,C 180,E1 -2977.766,E2 -2977.766} C_VEL
LIN {X 0,Y 559.227,Z 440.537,A -85,B 0,C 180,E1 -2978.401,E2 -2978.401} C_VEL
LIN {X 0,Y 559.292,Z 432.225,A -85,B 0,C 180,E1 -2978.946,E2 -2978.946} C_VEL
LIN {X 0,Y 559.385,Z 421.611,A -85,B 0,C 180,E1 -2979.491,E2 -2979.491} C_VEL
LIN {X 0,Y 559.5,Z 410.077,A -85,B 0,C 180,E1 -2979.9,E2 -2979.9} C_VEL
LIN {X 0,Y 559.578,Z 400.44,A -85,B 0,C 180,E1 -2980.127,E2 -2980.127} C_VEL
LIN {X 0,Y 559.745,Z 331.181,A -85,B 0,C 180,E1 -2981.032,E2 -2981.032} C_VEL
LIN {X 0,Y 559.357,Z 324.604,A -85,B 0,C 180,E1 -2981.124,E2 -2981.124} C_VEL
LIN {X 0,Y 559.091,Z 322.256,A -85,B 0,C 180,E1 -2981.172,E2 -2981.172} C_VEL
LIN {X 0,Y 559.336,Z 302.859,A -85,B 0,C 180,E1 -2984.183,E2 -2984.183} C_VEL
LIN {X 0,Y 559.478,Z 284.37,A -85,B 0,C 180,E1 -2987.053,E2 -2987.053} C_VEL
LIN {X 0,Y 559.643,Z 266.694,A -85,B 0,C 180,E1 -2989.82,E2 -2989.82} C_VEL
LIN {X 0,Y 559.923,Z 250.934,A -85,B 0,C 180,E1 -2992.314,E2 -2992.314} C_VEL
LIN {X 0,Y 559.139,Z 245.653,A -85,B 0,C 180,E1 -2993.221,E2 -2993.221} C_VEL
LIN {X 0,Y 559.172,Z 245.642,A -85,B 0,C 180,E1 -2996.097,E2 -2996.097} C_VEL
LIN {X 0,Y 559.138,Z 245.643,A -85,B 0,C 180,E1 -2998.531,E2 -2998.531} C_VEL
LIN {X 0,Y 559.144,Z 245.648,A -85,B 0,C 180,E1 -3001.273,E2 -3001.273} C_VEL
LIN {X 0,Y 559.165,Z 245.643,A -85,B 0,C 180,E1 -3003.949,E2 -3003.949} C_VEL
LIN {X 0,Y 559.142,Z 245.646,A -85,B 0,C 180,E1 -3007.108,E2 -3007.108} C_VEL
LIN {X 0,Y 559.158,Z 245.644,A -85,B 0,C 180,E1 -3009.941,E2 -3009.941} C_VEL
LIN {X 0,Y 559.159,Z 245.641,A -85,B 0,C 180,E1 -3012.743,E2 -3012.743} C_VEL
LIN {X 0,Y 559.15,Z 245.648,A -85,B 0,C 180,E1 -3015.76,E2 -3015.76} C_VEL
LIN {X 0,Y 559.183,Z 245.638,A -85,B 0,C 180,E1 -3018.231,E2 -3018.231} C_VEL
LIN {X 0,Y 559.173,Z 245.643,A -85,B 0,C 180,E1 -3021.191,E2 -3021.191} C_VEL
LIN {X 0,Y 559.157,Z 245.646,A -85,B 0,C 180,E1 -3023.79,E2 -3023.79} C_VEL
LIN {X 0,Y 559.158,Z 245.641,A -85,B 0,C 180,E1 -3026.424,E2 -3026.424} C_VEL
LIN {X 0,Y 559.151,Z 245.644,A -85,B 0,C 180,E1 -3028.98,E2 -3028.98} C_VEL
LIN {X 0,Y 559.166,Z 245.648,A -85,B 0,C 180,E1 -3031.618,E2 -3031.618} C_VEL
LIN {X 0,Y 559.195,Z 245.64,A -85,B 0,C 180,E1 -3033.903,E2 -3033.903} C_VEL
LIN {X 0,Y 559.152,Z 245.641,A -85,B 0,C 180,E1 -3036.567,E2 -3036.567} C_VEL
LIN {X 0,Y 559.175,Z 245.646,A -85,B 0,C 180,E1 -3039.395,E2 -3039.395} C_VEL
LIN {X 0,Y 559.143,Z 245.65,A -85,B 0,C 180,E1 -3041.685,E2 -3041.685} C_VEL
LIN {X 0,Y 559.162,Z 245.644,A -85,B 0,C 180,E1 -3043.947,E2 -3043.947} C_VEL
LIN {X 0,Y 559.166,Z 245.641,A -85,B 0,C 180,E1 -3046.183,E2 -3046.183} C_VEL
LIN {X 0,Y 559.19,Z 245.64,A -85,B 0,C 180,E1 -3049.133,E2 -3049.133} C_VEL
LIN {X 0,Y 559.202,Z 245.638,A -85,B 0,C 180,E1 -3052.053,E2 -3052.053} C_VEL
LIN {X 0,Y 559.25,Z 245.631,A -85,B 0,C 180,E1 -3054.953,E2 -3054.953} C_VEL
LIN {X 0,Y 559.245,Z 245.635,A -85,B 0,C 180,E1 -3057.839,E2 -3057.839} C_VEL
LIN {X 0,Y 559.269,Z 245.627,A -85,B 0,C 180,E1 -3060.719,E2 -3060.719} C_VEL
LIN {X 0,Y 559.237,Z 245.632,A -85,B 0,C 180,E1 -3062.881,E2 -3062.881} C_VEL
LIN {X 0,Y 559.221,Z 245.639,A -85,B 0,C 180,E1 -3065.77,E2 -3065.77} C_VEL
LIN {X 0,Y 559.186,Z 245.637,A -85,B 0,C 180,E1 -3068.674,E2 -3068.674} C_VEL
LIN {X 0,Y 559.197,Z 245.645,A -85,B 0,C 180,E1 -3071.6,E2 -3071.6} C_VEL
LIN {X 0,Y 559.191,Z 245.637,A -85,B 0,C 180,E1 -3074.595,E2 -3074.595} C_VEL
LIN {X 0,Y 559.156,Z 245.651,A -85,B 0,C 180,E1 -3077.556,E2 -3077.556} C_VEL
LIN {X 0,Y 559.166,Z 245.645,A -85,B 0,C 180,E1 -3079.837,E2 -3079.837} C_VEL
LIN {X 0,Y 559.134,Z 245.645,A -85,B 0,C 180,E1 -3082.152,E2 -3082.152} C_VEL
LIN {X 0,Y 559.17,Z 245.643,A -85,B 0,C 180,E1 -3085.187,E2 -3085.187} C_VEL
LIN {X 0,Y 559.185,Z 245.645,A -85,B 0,C 180,E1 -3087.711,E2 -3087.711} C_VEL
LIN {X 0,Y 559.136,Z 245.643,A -85,B 0,C 180,E1 -3090.628,E2 -3090.628} C_VEL
LIN {X 0,Y 558.478,Z 245.732,A -85,B 0,C 180,E1 -3091.229,E2 -3091.229} C_VEL
LIN {X 0,Y 555.618,Z 246.083,A -85,B 0,C 180,E1 -3092.205,E2 -3092.205} C_VEL
LIN {X 0,Y 553.207,Z 246.384,A -85,B 0,C 180,E1 -3092.991,E2 -3092.991} C_VEL
LIN {X 0,Y 552.188,Z 246.519,A -85,B 0,C 180,E1 -3093.598,E2 -3093.598} C_VEL
LIN {X 0,Y 552.115,Z 246.52,A -85,B 0,C 180,E1 -3093.803,E2 -3093.803} C_VEL
LIN {X 0,Y 552.102,Z 246.52,A -85,B 0,C 180,E1 -3096.746,E2 -3096.746} C_VEL
LIN {X 0,Y 552.14,Z 246.524,A -85,B 0,C 180,E1 -3099.525,E2 -3099.525} C_VEL
LIN {X 0,Y 552.121,Z 246.518,A -85,B 0,C 180,E1 -3102.425,E2 -3102.425} C_VEL
LIN {X 0,Y 552.09,Z 246.531,A -85,B 0,C 180,E1 -3105.563,E2 -3105.563} C_VEL
LIN {X 0,Y 552.131,Z 246.516,A -85,B 0,C 180,E1 -3108.676,E2 -3108.676} C_VEL
LIN {X 0,Y 552.11,Z 246.526,A -85,B 0,C 180,E1 -3111.411,E2 -3111.411} C_VEL
LIN {X 0,Y 552.091,Z 246.523,A -85,B 0,C 180,E1 -3114.157,E2 -3114.157} C_VEL
LIN {X 0,Y 552.114,Z 246.519,A -85,B 0,C 180,E1 -3116.815,E2 -3116.815} C_VEL
LIN {X 0,Y 552.098,Z 246.527,A -85,B 0,C 180,E1 -3119.391,E2 -3119.391} C_VEL
LIN {X 0,Y 552.117,Z 246.523,A -85,B 0,C 180,E1 -3121.903,E2 -3121.903} C_VEL
LIN {X 0,Y 552.146,Z 246.514,A -85,B 0,C 180,E1 -3124.649,E2 -3124.649} C_VEL
LIN {X 0,Y 552.105,Z 246.529,A -85,B 0,C 180,E1 -3127.55,E2 -3127.55} C_VEL
LIN {X 0,Y 552.148,Z 246.514,A -85,B 0,C 180,E1 -3130.674,E2 -3130.674} C_VEL
LIN {X 0,Y 552.111,Z 246.526,A -85,B 0,C 180,E1 -3133.737,E2 -3133.737} C_VEL
LIN {X 0,Y 552.127,Z 246.52,A -85,B 0,C 180,E1 -3136.004,E2 -3136.004} C_VEL
LIN {X 0,Y 552.169,Z 246.513,A -85,B 0,C 180,E1 -3138.994,E2 -3138.994} C_VEL
LIN {X 0,Y 552.15,Z 246.518,A -85,B 0,C 180,E1 -3141.951,E2 -3141.951} C_VEL
LIN {X 0,Y 552.22,Z 246.506,A -85,B 0,C 180,E1 -3144.889,E2 -3144.889} C_VEL
LIN {X 0,Y 552.209,Z 246.513,A -85,B 0,C 180,E1 -3147.812,E2 -3147.812} C_VEL
LIN {X 0,Y 552.231,Z 246.504,A -85,B 0,C 180,E1 -3150.729,E2 -3150.729} C_VEL
LIN {X 0,Y 552.195,Z 246.509,A -85,B 0,C 180,E1 -3152.918,E2 -3152.918} C_VEL
LIN {X 0,Y 552.179,Z 246.516,A -85,B 0,C 180,E1 -3155.844,E2 -3155.844} C_VEL
LIN {X 0,Y 552.135,Z 246.516,A -85,B 0,C 180,E1 -3158.786,E2 -3158.786} C_VEL
LIN {X 0,Y 552.152,Z 246.521,A -85,B 0,C 180,E1 -3161.75,E2 -3161.75} C_VEL
LIN {X 0,Y 552.118,Z 246.518,A -85,B 0,C 180,E1 -3164.748,E2 -3164.748} C_VEL
LIN {X 0,Y 552.095,Z 246.527,A -85,B 0,C 180,E1 -3167.788,E2 -3167.788} C_VEL
LIN {X 0,Y 552.117,Z 246.521,A -85,B 0,C 180,E1 -3170.101,E2 -3170.101} C_VEL
LIN {X 0,Y 552.079,Z 246.523,A -85,B 0,C 180,E1 -3172.451,E2 -3172.451} C_VEL
LIN {X 0,Y 552.103,Z 246.529,A -85,B 0,C 180,E1 -3175.645,E2 -3175.645} C_VEL
LIN {X 0,Y 552.078,Z 246.525,A -85,B 0,C 180,E1 -3178.099,E2 -3178.099} C_VEL
LIN {X 0,Y 552.089,Z 246.522,A -85,B 0,C 180,E1 -3180.609,E2 -3180.609} C_VEL
LIN {X 0,Y 552.049,Z 246.533,A -85,B 0,C 180,E1 -3183.257,E2 -3183.257} C_VEL
LIN {X 0,Y 551.911,Z 259.085,A -85,B 0,C 180,E1 -3186.255,E2 -3186.255} C_VEL
LIN {X 0,Y 551.847,Z 265.386,A -85,B 0,C 180,E1 -3187.767,E2 -3187.767} C_VEL
LIN {X 0,Y 552.766,Z 273.38,A -85,B 0,C 180,E1 -3187.899,E2 -3187.899} C_VEL
LIN {X 0,Y 552.568,Z 340.088,A -85,B 0,C 180,E1 -3188.781,E2 -3188.781} C_VEL
LIN {X 0,Y 552.427,Z 349.714,A -85,B 0,C 180,E1 -3189.005,E2 -3189.005} C_VEL
LIN {X 0,Y 552.367,Z 360.651,A -85,B 0,C 180,E1 -3189.39,E2 -3189.39} C_VEL
LIN {X 0,Y 552.258,Z 370.394,A -85,B 0,C 180,E1 -3189.87,E2 -3189.87} C_VEL
LIN {X 0,Y 552.16,Z 379.724,A -85,B 0,C 180,E1 -3190.475,E2 -3190.475} C_VEL
LIN {X 0,Y 552.118,Z 385.958,A -85,B 0,C 180,E1 -3190.96,E2 -3190.96} C_VEL
LIN {X 0,Y 551.979,Z 393.773,A -85,B 0,C 180,E1 -3191.701,E2 -3191.701} C_VEL
LIN {X 0,Y 551.895,Z 400.22,A -85,B 0,C 180,E1 -3192.446,E2 -3192.446} C_VEL
LIN {X 0,Y 551.836,Z 405.61,A -85,B 0,C 180,E1 -3193.198,E2 -3193.198} C_VEL
LIN {X 0,Y 551.785,Z 410.137,A -85,B 0,C 180,E1 -3193.959,E2 -3193.959} C_VEL
LIN {X 0,Y 551.771,Z 413.893,A -85,B 0,C 180,E1 -3194.725,E2 -3194.725} C_VEL
LIN {X 0,Y 551.72,Z 417.052,A -85,B 0,C 180,E1 -3195.526,E2 -3195.526} C_VEL
LIN {X 0,Y 551.698,Z 420.027,A -85,B 0,C 180,E1 -3196.56,E2 -3196.56} C_VEL
LIN {X 0,Y 551.647,Z 421.999,A -85,B 0,C 180,E1 -3197.638,E2 -3197.638} C_VEL
LIN {X 0,Y 551.655,Z 422.889,A -85,B 0,C 180,E1 -3198.732,E2 -3198.732} C_VEL
LIN {X 0,Y 551.636,Z 422.672,A -85,B 0,C 180,E1 -3199.854,E2 -3199.854} C_VEL
LIN {X 0,Y 551.657,Z 421.206,A -85,B 0,C 180,E1 -3200.997,E2 -3200.997} C_VEL
LIN {X 0,Y 551.718,Z 418.316,A -85,B 0,C 180,E1 -3202.163,E2 -3202.163} C_VEL
LIN {X 0,Y 551.747,Z 416.354,A -85,B 0,C 180,E1 -3202.769,E2 -3202.769} C_VEL
LIN {X 0,Y 551.789,Z 411.119,A -85,B 0,C 180,E1 -3203.943,E2 -3203.943} C_VEL
LIN {X 0,Y 551.835,Z 406.107,A -85,B 0,C 180,E1 -3204.815,E2 -3204.815} C_VEL
LIN {X 0,Y 551.88,Z 401.512,A -85,B 0,C 180,E1 -3205.477,E2 -3205.477} C_VEL
LIN {X 0,Y 551.955,Z 394.983,A -85,B 0,C 180,E1 -3206.258,E2 -3206.258} C_VEL
LIN {X 0,Y 552.067,Z 388.364,A -85,B 0,C 180,E1 -3206.913,E2 -3206.913} C_VEL
LIN {X 0,Y 552.17,Z 379.991,A -85,B 0,C 180,E1 -3207.594,E2 -3207.594} C_VEL
LIN {X 0,Y 552.309,Z 370.168,A -85,B 0,C 180,E1 -3208.232,E2 -3208.232} C_VEL
LIN {X 0,Y 552.372,Z 358.813,A -85,B 0,C 180,E1 -3208.771,E2 -3208.771} C_VEL
LIN {X 0,Y 552.502,Z 349.174,A -85,B 0,C 180,E1 -3209.098,E2 -3209.098} C_VEL
LIN {X 0,Y 552.559,Z 340.558,A -85,B 0,C 180,E1 -3209.301,E2 -3209.301} C_VEL
LIN {X 0,Y 552.76,Z 278.407,A -85,B 0,C 180,E1 -3210.126,E2 -3210.126} C_VEL
LIN {X 0,Y 552.591,Z 270.084,A -85,B 0,C 180,E1 -3210.237,E2 -3210.237} C_VEL
LIN {X 0,Y 551.881,Z 265.27,A -85,B 0,C 180,E1 -3210.327,E2 -3210.327} C_VEL
LIN {X 0,Y 551.924,Z 256.657,A -85,B 0,C 180,E1 -3212.305,E2 -3212.305} C_VEL
LIN {X 0,Y 551.949,Z 249.125,A -85,B 0,C 180,E1 -3213.942,E2 -3213.942} C_VEL
LIN {X 0,Y 551.981,Z 246.545,A -85,B 0,C 180,E1 -3214.546,E2 -3214.546} C_VEL
LIN {X 0,Y 552.091,Z 246.529,A -85,B 0,C 180,E1 -3216.758,E2 -3216.758} C_VEL
LIN {X 0,Y 552.115,Z 246.522,A -85,B 0,C 180,E1 -3219.121,E2 -3219.121} C_VEL
LIN {X 0,Y 552.121,Z 246.519,A -85,B 0,C 180,E1 -3221.445,E2 -3221.445} C_VEL
LIN {X 0,Y 552.11,Z 246.52,A -85,B 0,C 180,E1 -3223.738,E2 -3223.738} C_VEL
LIN {X 0,Y 552.126,Z 246.52,A -85,B 0,C 180,E1 -3226.005,E2 -3226.005} C_VEL
LIN {X 0,Y 552.168,Z 246.515,A -85,B 0,C 180,E1 -3228.994,E2 -3228.994} C_VEL
LIN {X 0,Y 552.154,Z 246.516,A -85,B 0,C 180,E1 -3231.952,E2 -3231.952} C_VEL
LIN {X 0,Y 552.225,Z 246.508,A -85,B 0,C 180,E1 -3234.89,E2 -3234.89} C_VEL
LIN {X 0,Y 552.214,Z 246.506,A -85,B 0,C 180,E1 -3237.813,E2 -3237.813} C_VEL
LIN {X 0,Y 552.237,Z 246.508,A -85,B 0,C 180,E1 -3240.73,E2 -3240.73} C_VEL
LIN {X 0,Y 552.202,Z 246.511,A -85,B 0,C 180,E1 -3242.919,E2 -3242.919} C_VEL
LIN {X 0,Y 552.192,Z 246.509,A -85,B 0,C 180,E1 -3245.845,E2 -3245.845} C_VEL
LIN {X 0,Y 552.162,Z 246.517,A -85,B 0,C 180,E1 -3248.786,E2 -3248.786} C_VEL
LIN {X 0,Y 552.154,Z 246.513,A -85,B 0,C 180,E1 -3251.751,E2 -3251.751} C_VEL
LIN {X 0,Y 552.128,Z 246.522,A -85,B 0,C 180,E1 -3254.749,E2 -3254.749} C_VEL
LIN {X 0,Y 552.107,Z 246.519,A -85,B 0,C 180,E1 -3257.789,E2 -3257.789} C_VEL
LIN {X 0,Y 552.126,Z 246.52,A -85,B 0,C 180,E1 -3260.102,E2 -3260.102} C_VEL
LIN {X 0,Y 552.089,Z 246.529,A -85,B 0,C 180,E1 -3262.452,E2 -3262.452} C_VEL
LIN {X 0,Y 552.15,Z 246.512,A -85,B 0,C 180,E1 -3265.352,E2 -3265.352} C_VEL
LIN {X 0,Y 552.12,Z 246.521,A -85,B 0,C 180,E1 -3268.098,E2 -3268.098} C_VEL
LIN {X 0,Y 552.104,Z 246.528,A -85,B 0,C 180,E1 -3270.61,E2 -3270.61} C_VEL
LIN {X 0,Y 552.117,Z 246.517,A -85,B 0,C 180,E1 -3273.186,E2 -3273.186} C_VEL
LIN {X 0,Y 552.107,Z 246.521,A -85,B 0,C 180,E1 -3275.842,E2 -3275.842} C_VEL
LIN {X 0,Y 552.12,Z 246.52,A -85,B 0,C 180,E1 -3279.063,E2 -3279.063} C_VEL
LIN {X 0,Y 552.132,Z 246.516,A -85,B 0,C 180,E1 -3281.445,E2 -3281.445} C_VEL
LIN {X 0,Y 552.09,Z 246.531,A -85,B 0,C 180,E1 -3284.533,E2 -3284.533} C_VEL
LIN {X 0,Y 552.127,Z 246.517,A -85,B 0,C 180,E1 -3287.585,E2 -3287.585} C_VEL
LIN {X 0,Y 552.126,Z 246.527,A -85,B 0,C 180,E1 -3290.474,E2 -3290.474} C_VEL
LIN {X 0,Y 552.109,Z 246.52,A -85,B 0,C 180,E1 -3293.317,E2 -3293.317} C_VEL
LIN {X 0,Y 552.125,Z 246.52,A -85,B 0,C 180,E1 -3295.94,E2 -3295.94} C_VEL
LIN {X 0,Y 552.117,Z 246.528,A -85,B 0,C 180,E1 -3298.541,E2 -3298.541} C_VEL
LIN {X 0,Y 552.102,Z 246.521,A -85,B 0,C 180,E1 -3301.443,E2 -3301.443} C_VEL
LIN {X 0,Y 552.126,Z 246.526,A -85,B 0,C 180,E1 -3304.356,E2 -3304.356} C_VEL
LIN {X 0,Y 552.148,Z 246.622,A -85,B 0,C 180,E1 -3306.909,E2 -3306.909} C_VEL
LIN {X 0,Y 552.755,Z 251.863,A -85,B 0,C 180,E1 -3307.748,E2 -3307.748} C_VEL
LIN {X 0,Y 552.57,Z 267.94,A -85,B 0,C 180,E1 -3310.252,E2 -3310.252} C_VEL
LIN {X 0,Y 552.422,Z 285.421,A -85,B 0,C 180,E1 -3312.986,E2 -3312.986} C_VEL
LIN {X 0,Y 552.26,Z 304.922,A -85,B 0,C 180,E1 -3316.008,E2 -3316.008} C_VEL
LIN {X 0,Y 552.053,Z 322.293,A -85,B 0,C 180,E1 -3318.689,E2 -3318.689} C_VEL
LIN {X 0,Y 552.761,Z 329.37,A -85,B 0,C 180,E1 -3318.803,E2 -3318.803} C_VEL
LIN {X 0,Y 552.631,Z 399.161,A -85,B 0,C 180,E1 -3319.721,E2 -3319.721} C_VEL
LIN {X 0,Y 552.517,Z 408.424,A -85,B 0,C 180,E1 -3319.928,E2 -3319.928} C_VEL
LIN {X 0,Y 552.402,Z 418.102,A -85,B 0,C 180,E1 -3320.249,E2 -3320.249} C_VEL
LIN {X 0,Y 552.342,Z 427.269,A -85,B 0,C 180,E1 -3320.664,E2 -3320.664} C_VEL
LIN {X 0,Y 552.256,Z 438.075,A -85,B 0,C 180,E1 -3321.308,E2 -3321.308} C_VEL
LIN {X 0,Y 552.073,Z 447.375,A -85,B 0,C 180,E1 -3322.043,E2 -3322.043} C_VEL
LIN {X 0,Y 551.994,Z 454.038,A -85,B 0,C 180,E1 -3322.686,E2 -3322.686} C_VEL
LIN {X 0,Y 551.949,Z 460.359,A -85,B 0,C 180,E1 -3323.42,E2 -3323.42} C_VEL
LIN {X 0,Y 551.917,Z 465.612,A -85,B 0,C 180,E1 -3324.153,E2 -3324.153} C_VEL
LIN {X 0,Y 551.743,Z 469.99,A -85,B 0,C 180,E1 -3324.885,E2 -3324.885} C_VEL
LIN {X 0,Y 551.779,Z 475.15,A -85,B 0,C 180,E1 -3325.983,E2 -3325.983} C_VEL
LIN {X 0,Y 551.729,Z 478.938,A -85,B 0,C 180,E1 -3327.08,E2 -3327.08} C_VEL
LIN {X 0,Y 551.657,Z 480.682,A -85,B 0,C 180,E1 -3327.81,E2 -3327.81} C_VEL
LIN {X 0,Y 551.644,Z 481.93,A -85,B 0,C 180,E1 -3328.54,E2 -3328.54} C_VEL
LIN {X 0,Y 551.638,Z 482.707,A -85,B 0,C 180,E1 -3329.27,E2 -3329.27} C_VEL
LIN {X 0,Y 551.637,Z 483,A -85,B 0,C 180,E1 -3330,E2 -3330} C_VEL
LIN {X 0,Y 551.638,Z 482.707,A -85,B 0,C 180,E1 -3330.73,E2 -3330.73} C_VEL
LIN {X 0,Y 551.644,Z 481.929,A -85,B 0,C 180,E1 -3331.46,E2 -3331.46} C_VEL
LIN {X 0,Y 551.657,Z 480.68,A -85,B 0,C 180,E1 -3332.19,E2 -3332.19} C_VEL
LIN {X 0,Y 551.761,Z 477.786,A -85,B 0,C 180,E1 -3333.286,E2 -3333.286} C_VEL
LIN {X 0,Y 551.779,Z 475.148,A -85,B 0,C 180,E1 -3334.017,E2 -3334.017} C_VEL
LIN {X 0,Y 551.743,Z 469.985,A -85,B 0,C 180,E1 -3335.116,E2 -3335.116} C_VEL
LIN {X 0,Y 551.957,Z 463.4,A -85,B 0,C 180,E1 -3336.184,E2 -3336.184} C_VEL
LIN {X 0,Y 551.993,Z 455.741,A -85,B 0,C 180,E1 -3337.131,E2 -3337.131} C_VEL
LIN {X 0,Y 552.076,Z 448.398,A -85,B 0,C 180,E1 -3337.866,E2 -3337.866} C_VEL
LIN {X 0,Y 552.202,Z 440.534,A -85,B 0,C 180,E1 -3338.508,E2 -3338.508} C_VEL
LIN {X 0,Y 552.26,Z 432.222,A -85,B 0,C 180,E1 -3339.061,E2 -3339.061} C_VEL
LIN {X 0,Y 552.393,Z 421.61,A -85,B 0,C 180,E1 -3339.613,E2 -3339.613} C_VEL
LIN {X 0,Y 552.511,Z 410.076,A -85,B 0,C 180,E1 -3340.027,E2 -3340.027} C_VEL
LIN {X 0,Y 552.615,Z 400.439,A -85,B 0,C 180,E1 -3340.256,E2 -3340.256} C_VEL
LIN {X 0,Y 552.776,Z 330.898,A -85,B 0,C 180,E1 -3341.177,E2 -3341.177} C_VEL
LIN {X 0,Y 552.257,Z 323.967,A -85,B 0,C 180,E1 -3341.277,E2 -3341.277} C_VEL
LIN {X 0,Y 552.05,Z 322.303,A -85,B 0,C 180,E1 -3341.309,E2 -3341.309} C_VEL
LIN {X 0,Y 552.29,Z 303.877,A -85,B 0,C 180,E1 -3344.173,E2 -3344.173} C_VEL
LIN {X 0,Y 552.447,Z 285.753,A -85,B 0,C 180,E1 -3347.013,E2 -3347.013} C_VEL
LIN {X 0,Y 552.626,Z 268.386,A -85,B 0,C 180,E1 -3349.764,E2 -3349.764} C_VEL
LIN {X 0,Y 552.92,Z 252.827,A -85,B 0,C 180,E1 -3352.252,E2 -3352.252} C_VEL
LIN {X 0,Y 552.404,Z 248.137,A -85,B 0,C 180,E1 -3353.03,E2 -3353.03} C_VEL
LIN {X 0,Y 552.096,Z 246.53,A -85,B 0,C 180,E1 -3353.325,E2 -3353.325} C_VEL
LIN {X 0,Y 552.127,Z 246.526,A -85,B 0,C 180,E1 -3355.644,E2 -3355.644} C_VEL
LIN {X 0,Y 552.104,Z 246.52,A -85,B 0,C 180,E1 -3358.558,E2 -3358.558} C_VEL
LIN {X 0,Y 552.111,Z 246.528,A -85,B 0,C 180,E1 -3361.475,E2 -3361.475} C_VEL
LIN {X 0,Y 552.133,Z 246.517,A -85,B 0,C 180,E1 -3364.17,E2 -3364.17} C_VEL
LIN {X 0,Y 552.108,Z 246.519,A -85,B 0,C 180,E1 -3366.746,E2 -3366.746} C_VEL
LIN {X 0,Y 552.127,Z 246.527,A -85,B 0,C 180,E1 -3369.527,E2 -3369.527} C_VEL
LIN {X 0,Y 552.129,Z 246.516,A -85,B 0,C 180,E1 -3372.425,E2 -3372.425} C_VEL
LIN {X 0,Y 552.096,Z 246.53,A -85,B 0,C 180,E1 -3375.562,E2 -3375.562} C_VEL
LIN {X 0,Y 552.135,Z 246.516,A -85,B 0,C 180,E1 -3378.676,E2 -3378.676} C_VEL
LIN {X 0,Y 552.115,Z 246.526,A -85,B 0,C 180,E1 -3381.411,E2 -3381.411} C_VEL
LIN {X 0,Y 552.099,Z 246.521,A -85,B 0,C 180,E1 -3384.157,E2 -3384.157} C_VEL
LIN {X 0,Y 552.111,Z 246.519,A -85,B 0,C 180,E1 -3386.814,E2 -3386.814} C_VEL
LIN {X 0,Y 552.098,Z 246.528,A -85,B 0,C 180,E1 -3389.39,E2 -3389.39} C_VEL
LIN {X 0,Y 552.123,Z 246.521,A -85,B 0,C 180,E1 -3391.902,E2 -3391.902} C_VEL
LIN {X 0,Y 552.153,Z 246.513,A -85,B 0,C 180,E1 -3394.648,E2 -3394.648} C_VEL
LIN {X 0,Y 552.091,Z 246.531,A -85,B 0,C 180,E1 -3397.549,E2 -3397.549} C_VEL
LIN {X 0,Y 552.143,Z 246.515,A -85,B 0,C 180,E1 -3400.373,E2 -3400.373} C_VEL
LIN {X 0,Y 552.15,Z 246.516,A -85,B 0,C 180,E1 -3402.977,E2 -3402.977} C_VEL
LIN {X 0,Y 552.13,Z 246.519,A -85,B 0,C 180,E1 -3406.004,E2 -3406.004} C_VEL
LIN {X 0,Y 552.157,Z 246.515,A -85,B 0,C 180,E1 -3408.993,E2 -3408.993} C_VEL
LIN {X 0,Y 552.157,Z 246.516,A -85,B 0,C 180,E1 -3411.951,E2 -3411.951} C_VEL
LIN {X 0,Y 552.224,Z 246.506,A -85,B 0,C 180,E1 -3414.888,E2 -3414.888} C_VEL
LIN {X 0,Y 552.217,Z 246.511,A -85,B 0,C 180,E1 -3417.811,E2 -3417.811} C_VEL
LIN {X 0,Y 552.239,Z 246.503,A -85,B 0,C 180,E1 -3420.729,E2 -3420.729} C_VEL
LIN {X 0,Y 552.203,Z 246.508,A -85,B 0,C 180,E1 -3422.917,E2 -3422.917} C_VEL
LIN {X 0,Y 552.191,Z 246.514,A -85,B 0,C 180,E1 -3425.843,E2 -3425.843} C_VEL
LIN {X 0,Y 552.156,Z 246.513,A -85,B 0,C 180,E1 -3428.785,E2 -3428.785} C_VEL
LIN {X 0,Y 552.154,Z 246.52,A -85,B 0,C 180,E1 -3431.75,E2 -3431.75} C_VEL
LIN {X 0,Y 552.128,Z 246.517,A -85,B 0,C 180,E1 -3434.748,E2 -3434.748} C_VEL
LIN {X 0,Y 552.107,Z 246.525,A -85,B 0,C 180,E1 -3437.788,E2 -3437.788} C_VEL
LIN {X 0,Y 552.126,Z 246.519,A -85,B 0,C 180,E1 -3440.101,E2 -3440.101} C_VEL
LIN {X 0,Y 552.087,Z 246.522,A -85,B 0,C 180,E1 -3442.45,E2 -3442.45} C_VEL
LIN {X 0,Y 552.148,Z 246.521,A -85,B 0,C 180,E1 -3445.35,E2 -3445.35} C_VEL
LIN {X 0,Y 552.117,Z 246.52,A -85,B 0,C 180,E1 -3448.097,E2 -3448.097} C_VEL
LIN {X 0,Y 552.097,Z 246.52,A -85,B 0,C 180,E1 -3450.623,E2 -3450.623} C_VEL
LIN {X 0,Y 552.12,Z 246.522,A -85,B 0,C 180,E1 -3453.184,E2 -3453.184} C_VEL
LIN {X 0,Y 552.115,Z 246.52,A -85,B 0,C 180,E1 -3453.803,E2 -3453.803} C_VEL
LIN {X 0,Y 551.48,Z 246.601,A -85,B 0,C 180,E1 -3454.412,E2 -3454.412} C_VEL
LIN {X 0,Y 548.654,Z 246.956,A -85,B 0,C 180,E1 -3455.4,E2 -3455.4} C_VEL
LIN {X 0,Y 546.228,Z 247.254,A -85,B 0,C 180,E1 -3456.195,E2 -3456.195} C_VEL
LIN {X 0,Y 545.157,Z 247.386,A -85,B 0,C 180,E1 -3456.809,E2 -3456.809} C_VEL
LIN {X 0,Y 545.055,Z 247.4,A -85,B 0,C 180,E1 -3457.017,E2 -3457.017} C_VEL
LIN {X 0,Y 545.066,Z 247.398,A -85,B 0,C 180,E1 -3460.141,E2 -3460.141} C_VEL
LIN {X 0,Y 545.076,Z 247.398,A -85,B 0,C 180,E1 -3463.105,E2 -3463.105} C_VEL
LIN {X 0,Y 545.056,Z 247.399,A -85,B 0,C 180,E1 -3466.224,E2 -3466.224} C_VEL
LIN {X 0,Y 545.092,Z 247.394,A -85,B 0,C 180,E1 -3468.887,E2 -3468.887} C_VEL
LIN {X 0,Y 545.045,Z 247.406,A -85,B 0,C 180,E1 -3471.763,E2 -3471.763} C_VEL
LIN {X 0,Y 545.043,Z 247.399,A -85,B 0,C 180,E1 -3474.533,E2 -3474.533} C_VEL
LIN {X 0,Y 545.073,Z 247.4,A -85,B 0,C 180,E1 -3477.212,E2 -3477.212} C_VEL
LIN {X 0,Y 545.057,Z 247.403,A -85,B 0,C 180,E1 -3479.811,E2 -3479.811} C_VEL
LIN {X 0,Y 545.084,Z 247.395,A -85,B 0,C 180,E1 -3482.344,E2 -3482.344} C_VEL
LIN {X 0,Y 545.108,Z 247.392,A -85,B 0,C 180,E1 -3484.82,E2 -3484.82} C_VEL
LIN {X 0,Y 545.057,Z 247.402,A -85,B 0,C 180,E1 -3487.243,E2 -3487.243} C_VEL
LIN {X 0,Y 545.112,Z 247.391,A -85,B 0,C 180,E1 -3490.415,E2 -3490.415} C_VEL
LIN {X 0,Y 545.068,Z 247.405,A -85,B 0,C 180,E1 -3493.521,E2 -3493.521} C_VEL
LIN {X 0,Y 545.086,Z 247.4,A -85,B 0,C 180,E1 -3495.82,E2 -3495.82} C_VEL
LIN {X 0,Y 545.123,Z 247.39,A -85,B 0,C 180,E1 -3498.85,E2 -3498.85} C_VEL
LIN {X 0,Y 545.12,Z 247.395,A -85,B 0,C 180,E1 -3501.847,E2 -3501.847} C_VEL
LIN {X 0,Y 545.195,Z 247.381,A -85,B 0,C 180,E1 -3504.823,E2 -3504.823} C_VEL
LIN {X 0,Y 545.181,Z 247.389,A -85,B 0,C 180,E1 -3507.783,E2 -3507.783} C_VEL
LIN {X 0,Y 545.201,Z 247.38,A -85,B 0,C 180,E1 -3510.738,E2 -3510.738} C_VEL
LIN {X 0,Y 545.162,Z 247.386,A -85,B 0,C 180,E1 -3512.956,E2 -3512.956} C_VEL
LIN {X 0,Y 545.15,Z 247.391,A -85,B 0,C 180,E1 -3515.919,E2 -3515.919} C_VEL
LIN {X 0,Y 545.097,Z 247.394,A -85,B 0,C 180,E1 -3518.9,E2 -3518.9} C_VEL
LIN {X 0,Y 545.124,Z 247.394,A -85,B 0,C 180,E1 -3521.904,E2 -3521.904} C_VEL
LIN {X 0,Y 545.071,Z 247.397,A -85,B 0,C 180,E1 -3524.943,E2 -3524.943} C_VEL
LIN {X 0,Y 545.057,Z 247.401,A -85,B 0,C 180,E1 -3528.026,E2 -3528.026} C_VEL
LIN {X 0,Y 545.082,Z 247.395,A -85,B 0,C 180,E1 -3530.372,E2 -3530.372} C_VEL
LIN {X 0,Y 545.064,Z 247.405,A -85,B 0,C 180,E1 -3533.559,E2 -3533.559} C_VEL
LIN {X 0,Y 545.058,Z 247.401,A -85,B 0,C 180,E1 -3536.001,E2 -3536.001} C_VEL
LIN {X 0,Y 545.062,Z 247.397,A -85,B 0,C 180,E1 -3538.745,E2 -3538.745} C_VEL
LIN {X 0,Y 545.046,Z 247.408,A -85,B 0,C 180,E1 -3541.679,E2 -3541.679} C_VEL
LIN {X 0,Y 544.972,Z 247.443,A -85,B 0,C 180,E1 -3543.295,E2 -3543.295} C_VEL
LIN {X 0,Y 544.868,Z 258.811,A -85,B 0,C 180,E1 -3545.991,E2 -3545.991} C_VEL
LIN {X 0,Y 544.812,Z 265.582,A -85,B 0,C 180,E1 -3547.612,E2 -3547.612} C_VEL
LIN {X 0,Y 545.802,Z 273.272,A -85,B 0,C 180,E1 -3547.75,E2 -3547.75} C_VEL
LIN {X 0,Y 545.59,Z 340.187,A -85,B 0,C 180,E1 -3548.647,E2 -3548.647} C_VEL
LIN {X 0,Y 545.457,Z 349.595,A -85,B 0,C 180,E1 -3548.866,E2 -3548.866} C_VEL
LIN {X 0,Y 545.414,Z 359.56,A -85,B 0,C 180,E1 -3549.212,E2 -3549.212} C_VEL
LIN {X 0,Y 545.261,Z 370.034,A -85,B 0,C 180,E1 -3549.713,E2 -3549.713} C_VEL
LIN {X 0,Y 545.185,Z 379.266,A -85,B 0,C 180,E1 -3550.306,E2 -3550.306} C_VEL
LIN {X 0,Y 545.058,Z 387.206,A -85,B 0,C 180,E1 -3550.942,E2 -3550.942} C_VEL
LIN {X 0,Y 544.92,Z 394.675,A -85,B 0,C 180,E1 -3551.676,E2 -3551.676} C_VEL
LIN {X 0,Y 544.83,Z 400.734,A -85,B 0,C 180,E1 -3552.397,E2 -3552.397} C_VEL
LIN {X 0,Y 544.784,Z 405.894,A -85,B 0,C 180,E1 -3553.134,E2 -3553.134} C_VEL
LIN {X 0,Y 544.707,Z 411.705,A -85,B 0,C 180,E1 -3554.164,E2 -3554.164} C_VEL
LIN {X 0,Y 544.648,Z 416.249,A -85,B 0,C 180,E1 -3555.21,E2 -3555.21} C_VEL
LIN {X 0,Y 544.614,Z 419.577,A -85,B 0,C 180,E1 -3556.273,E2 -3556.273} C_VEL
LIN {X 0,Y 544.56,Z 421.758,A -85,B 0,C 180,E1 -3557.359,E2 -3557.359} C_VEL
LIN {X 0,Y 544.583,Z 422.861,A -85,B 0,C 180,E1 -3558.46,E2 -3558.46} C_VEL
LIN {X 0,Y 544.539,Z 422.787,A -85,B 0,C 180,E1 -3559.812,E2 -3559.812} C_VEL
LIN {X 0,Y 544.555,Z 421.706,A -85,B 0,C 180,E1 -3560.775,E2 -3560.775} C_VEL
LIN {X 0,Y 544.633,Z 419.317,A -85,B 0,C 180,E1 -3561.918,E2 -3561.918} C_VEL
LIN {X 0,Y 544.675,Z 417.012,A -85,B 0,C 180,E1 -3562.668,E2 -3562.668} C_VEL
LIN {X 0,Y 544.72,Z 412.344,A -85,B 0,C 180,E1 -3563.803,E2 -3563.803} C_VEL
LIN {X 0,Y 544.774,Z 407.267,A -85,B 0,C 180,E1 -3564.74,E2 -3564.74} C_VEL
LIN {X 0,Y 544.841,Z 401.14,A -85,B 0,C 180,E1 -3565.642,E2 -3565.642} C_VEL
LIN {X 0,Y 544.913,Z 395.564,A -85,B 0,C 180,E1 -3566.319,E2 -3566.319} C_VEL
LIN {X 0,Y 545.044,Z 389.474,A -85,B 0,C 180,E1 -3566.941,E2 -3566.941} C_VEL
LIN {X 0,Y 545.168,Z 382.38,A -85,B 0,C 180,E1 -3567.548,E2 -3567.548} C_VEL
LIN {X 0,Y 545.285,Z 374.512,A -85,B 0,C 180,E1 -3568.101,E2 -3568.101} C_VEL
LIN {X 0,Y 545.336,Z 365.808,A -85,B 0,C 180,E1 -3568.593,E2 -3568.593} C_VEL
LIN {X 0,Y 545.42,Z 357.055,A -85,B 0,C 180,E1 -3568.976,E2 -3568.976} C_VEL
LIN {X 0,Y 545.528,Z 347.354,A -85,B 0,C 180,E1 -3569.287,E2 -3569.287} C_VEL
LIN {X 0,Y 545.61,Z 335.086,A -85,B 0,C 180,E1 -3569.529,E2 -3569.529} C_VEL
LIN {X 0,Y 545.775,Z 271.723,A -85,B 0,C 180,E1 -3570.36,E2 -3570.36} C_VEL
LIN {X 0,Y 544.83,Z 265.487,A -85,B 0,C 180,E1 -3570.463,E2 -3570.463} C_VEL
LIN {X 0,Y 544.848,Z 255.721,A -85,B 0,C 180,E1 -3572.633,E2 -3572.633} C_VEL
LIN {X 0,Y 544.918,Z 247.425,A -85,B 0,C 180,E1 -3574.408,E2 -3574.408} C_VEL
LIN {X 0,Y 545.075,Z 247.405,A -85,B 0,C 180,E1 -3576.441,E2 -3576.441} C_VEL
LIN {X 0,Y 545.088,Z 247.396,A -85,B 0,C 180,E1 -3579.629,E2 -3579.629} C_VEL
LIN {X 0,Y 545.084,Z 247.401,A -85,B 0,C 180,E1 -3582.75,E2 -3582.75} C_VEL
LIN {X 0,Y 545.084,Z 247.396,A -85,B 0,C 180,E1 -3585.82,E2 -3585.82} C_VEL
LIN {X 0,Y 545.122,Z 247.394,A -85,B 0,C 180,E1 -3588.85,E2 -3588.85} C_VEL
LIN {X 0,Y 545.124,Z 247.391,A -85,B 0,C 180,E1 -3591.848,E2 -3591.848} C_VEL
LIN {X 0,Y 545.2,Z 247.384,A -85,B 0,C 180,E1 -3594.824,E2 -3594.824} C_VEL
LIN {X 0,Y 545.186,Z 247.381,A -85,B 0,C 180,E1 -3597.784,E2 -3597.784} C_VEL
LIN {X 0,Y 545.207,Z 247.384,A -85,B 0,C 180,E1 -3600.739,E2 -3600.739} C_VEL
LIN {X 0,Y 545.168,Z 247.386,A -85,B 0,C 180,E1 -3602.956,E2 -3602.956} C_VEL
LIN {X 0,Y 545.163,Z 247.386,A -85,B 0,C 180,E1 -3605.92,E2 -3605.92} C_VEL
LIN {X 0,Y 545.119,Z 247.393,A -85,B 0,C 180,E1 -3608.901,E2 -3608.901} C_VEL
LIN {X 0,Y 545.126,Z 247.39,A -85,B 0,C 180,E1 -3611.905,E2 -3611.905} C_VEL
LIN {X 0,Y 545.077,Z 247.398,A -85,B 0,C 180,E1 -3614.944,E2 -3614.944} C_VEL
LIN {X 0,Y 545.075,Z 247.397,A -85,B 0,C 180,E1 -3618.026,E2 -3618.026} C_VEL
LIN {X 0,Y 545.091,Z 247.401,A -85,B 0,C 180,E1 -3620.373,E2 -3620.373} C_VEL
LIN {X 0,Y 545.084,Z 247.394,A -85,B 0,C 180,E1 -3623.56,E2 -3623.56} C_VEL
LIN {X 0,Y 545.082,Z 247.395,A -85,B 0,C 180,E1 -3626.001,E2 -3626.001} C_VEL
LIN {X 0,Y 545.086,Z 247.397,A -85,B 0,C 180,E1 -3628.75,E2 -3628.75} C_VEL
LIN {X 0,Y 545.062,Z 247.399,A -85,B 0,C 180,E1 -3631.048,E2 -3631.048} C_VEL
LIN {X 0,Y 545.065,Z 247.395,A -85,B 0,C 180,E1 -3633.672,E2 -3633.672} C_VEL
LIN {X 0,Y 545.055,Z 247.406,A -85,B 0,C 180,E1 -3636.38,E2 -3636.38} C_VEL
LIN {X 0,Y 545.1,Z 247.392,A -85,B 0,C 180,E1 -3639.325,E2 -3639.325} C_VEL
LIN {X 0,Y 545.077,Z 247.399,A -85,B 0,C 180,E1 -3642.103,E2 -3642.103} C_VEL
LIN {X 0,Y 545.057,Z 247.399,A -85,B 0,C 180,E1 -3645.168,E2 -3645.168} C_VEL
LIN {X 0,Y 545.077,Z 247.397,A -85,B 0,C 180,E1 -3647.898,E2 -3647.898} C_VEL
LIN {X 0,Y 545.076,Z 247.4,A -85,B 0,C 180,E1 -3650.819,E2 -3650.819} C_VEL
LIN {X 0,Y 545.047,Z 247.399,A -85,B 0,C 180,E1 -3653.621,E2 -3653.621} C_VEL
LIN {X 0,Y 545.067,Z 247.404,A -85,B 0,C 180,E1 -3656.329,E2 -3656.329} C_VEL
LIN {X 0,Y 545.064,Z 247.401,A -85,B 0,C 180,E1 -3658.953,E2 -3658.953} C_VEL
LIN {X 0,Y 545.081,Z 247.396,A -85,B 0,C 180,E1 -3661.507,E2 -3661.507} C_VEL
LIN {X 0,Y 545.084,Z 247.404,A -85,B 0,C 180,E1 -3664.494,E2 -3664.494} C_VEL
LIN {X 0,Y 545.111,Z 247.572,A -85,B 0,C 180,E1 -3666.845,E2 -3666.845} C_VEL
LIN {X 0,Y 545.746,Z 252.925,A -85,B 0,C 180,E1 -3667.713,E2 -3667.713} C_VEL
LIN {X 0,Y 545.532,Z 268.294,A -85,B 0,C 180,E1 -3670.127,E2 -3670.127} C_VEL
LIN {X 0,Y 545.369,Z 283.161,A -85,B 0,C 180,E1 -3672.481,E2 -3672.481} C_VEL
LIN {X 0,Y 545.264,Z 301.005,A -85,B 0,C 180,E1 -3675.287,E2 -3675.287} C_VEL
LIN {X 0,Y 545.013,Z 320.699,A -85,B 0,C 180,E1 -3678.36,E2 -3678.36} C_VEL
LIN {X 0,Y 544.971,Z 321.982,A -85,B 0,C 180,E1 -3678.552,E2 -3678.552} C_VEL
LIN {X 0,Y 545.809,Z 330.551,A -85,B 0,C 180,E1 -3678.681,E2 -3678.681} C_VEL
LIN {X 0,Y 545.623,Z 400.057,A -85,B 0,C 180,E1 -3679.611,E2 -3679.611} C_VEL
LIN {X 0,Y 545.502,Z 410.596,A -85,B 0,C 180,E1 -3679.867,E2 -3679.867} C_VEL
LIN {X 0,Y 545.374,Z 421.372,A -85,B 0,C 180,E1 -3680.263,E2 -3680.263} C_VEL
LIN {X 0,Y 545.247,Z 432.053,A -85,B 0,C 180,E1 -3680.822,E2 -3680.822} C_VEL
LIN {X 0,Y 545.156,Z 440.418,A -85,B 0,C 180,E1 -3681.381,E2 -3681.381} C_VEL
LIN {X 0,Y 545.009,Z 448.332,A -85,B 0,C 180,E1 -3682.032,E2 -3682.032} C_VEL
LIN {X 0,Y 544.92,Z 455.73,A -85,B 0,C 180,E1 -3682.777,E2 -3682.777} C_VEL
LIN {X 0,Y 544.869,Z 462.001,A -85,B 0,C 180,E1 -3683.549,E2 -3683.549} C_VEL
LIN {X 0,Y 544.711,Z 469.033,A -85,B 0,C 180,E1 -3684.633,E2 -3684.633} C_VEL
LIN {X 0,Y 544.707,Z 473.633,A -85,B 0,C 180,E1 -3685.56,E2 -3685.56} C_VEL
LIN {X 0,Y 544.676,Z 476.622,A -85,B 0,C 180,E1 -3686.301,E2 -3686.301} C_VEL
LIN {X 0,Y 544.659,Z 478.939,A -85,B 0,C 180,E1 -3687.042,E2 -3687.042} C_VEL
LIN {X 0,Y 544.572,Z 480.681,A -85,B 0,C 180,E1 -3687.781,E2 -3687.781} C_VEL
LIN {X 0,Y 544.545,Z 481.929,A -85,B 0,C 180,E1 -3688.521,E2 -3688.521} C_VEL
LIN {X 0,Y 544.538,Z 482.706,A -85,B 0,C 180,E1 -3689.261,E2 -3689.261} C_VEL
LIN {X 0,Y 544.538,Z 483,A -85,B 0,C 180,E1 -3690,E2 -3690} C_VEL
LIN {X 0,Y 544.538,Z 482.706,A -85,B 0,C 180,E1 -3690.74,E2 -3690.74} C_VEL
LIN {X 0,Y 544.545,Z 481.928,A -85,B 0,C 180,E1 -3691.479,E2 -3691.479} C_VEL
LIN {X 0,Y 544.572,Z 480.679,A -85,B 0,C 180,E1 -3692.219,E2 -3692.219} C_VEL
LIN {X 0,Y 544.689,Z 477.786,A -85,B 0,C 180,E1 -3693.329,E2 -3693.329} C_VEL
LIN {X 0,Y 544.702,Z 475.148,A -85,B 0,C 180,E1 -3694.069,E2 -3694.069} C_VEL
LIN {X 0,Y 544.671,Z 469.985,A -85,B 0,C 180,E1 -3695.182,E2 -3695.182} C_VEL
LIN {X 0,Y 544.88,Z 463.959,A -85,B 0,C 180,E1 -3696.182,E2 -3696.182} C_VEL
LIN {X 0,Y 544.921,Z 457.433,A -85,B 0,C 180,E1 -3697.037,E2 -3697.037} C_VEL
LIN {X 0,Y 545.016,Z 449.365,A -85,B 0,C 180,E1 -3697.875,E2 -3697.875} C_VEL
LIN {X 0,Y 545.145,Z 441.66,A -85,B 0,C 180,E1 -3698.526,E2 -3698.526} C_VEL
LIN {X 0,Y 545.25,Z 433.569,A -85,B 0,C 180,E1 -3699.085,E2 -3699.085} C_VEL
LIN {X 0,Y 545.34,Z 425.187,A -85,B 0,C 180,E1 -3699.551,E2 -3699.551} C_VEL
LIN {X 0,Y 545.443,Z 416.636,A -85,B 0,C 180,E1 -3699.924,E2 -3699.924} C_VEL
LIN {X 0,Y 545.533,Z 407.278,A -85,B 0,C 180,E1 -3700.227,E2 -3700.227} C_VEL
LIN {X 0,Y 545.663,Z 396.177,A -85,B 0,C 180,E1 -3700.459,E2 -3700.459} C_VEL
LIN {X 0,Y 545.654,Z 327.544,A -85,B 0,C 180,E1 -3701.362,E2 -3701.362} C_VEL
LIN {X 0,Y 544.996,Z 321.987,A -85,B 0,C 180,E1 -3701.461,E2 -3701.461} C_VEL
LIN {X 0,Y 545.267,Z 303.7,A -85,B 0,C 180,E1 -3704.338,E2 -3704.338} C_VEL
LIN {X 0,Y 545.436,Z 285.423,A -85,B 0,C 180,E1 -3707.239,E2 -3707.239} C_VEL
LIN {X 0,Y 545.697,Z 267.762,A -85,B 0,C 180,E1 -3710.071,E2 -3710.071} C_VEL
LIN {X 0,Y 545.94,Z 252.679,A -85,B 0,C 180,E1 -3712.519,E2 -3712.519} C_VEL
LIN {X 0,Y 545.078,Z 247.405,A -85,B 0,C 180,E1 -3713.458,E2 -3713.458} C_VEL
LIN {X 0,Y 545.075,Z 247.399,A -85,B 0,C 180,E1 -3716,E2 -3716} C_VEL
LIN {X 0,Y 545.074,Z 247.396,A -85,B 0,C 180,E1 -3718.745,E2 -3718.745} C_VEL
LIN {X 0,Y 545.057,Z 247.404,A -85,B 0,C 180,E1 -3721.678,E2 -3721.678} C_VEL
LIN {X 0,Y 545.066,Z 247.396,A -85,B 0,C 180,E1 -3724.564,E2 -3724.564} C_VEL
LIN {X 0,Y 545.036,Z 247.406,A -85,B 0,C 180,E1 -3727.303,E2 -3727.303} C_VEL
LIN {X 0,Y 545.064,Z 247.398,A -85,B 0,C 180,E1 -3730.142,E2 -3730.142} C_VEL
LIN {X 0,Y 545.077,Z 247.398,A -85,B 0,C 180,E1 -3733.106,E2 -3733.106} C_VEL
LIN {X 0,Y 545.048,Z 247.399,A -85,B 0,C 180,E1 -3736.225,E2 -3736.225} C_VEL
LIN {X 0,Y 545.096,Z 247.393,A -85,B 0,C 180,E1 -3738.886,E2 -3738.886} C_VEL
LIN {X 0,Y 545.05,Z 247.404,A -85,B 0,C 180,E1 -3741.762,E2 -3741.762} C_VEL
LIN {X 0,Y 545.049,Z 247.398,A -85,B 0,C 180,E1 -3744.532,E2 -3744.532} C_VEL
LIN {X 0,Y 545.065,Z 247.401,A -85,B 0,C 180,E1 -3747.211,E2 -3747.211} C_VEL
LIN {X 0,Y 545.059,Z 247.402,A -85,B 0,C 180,E1 -3749.81,E2 -3749.81} C_VEL
LIN {X 0,Y 545.092,Z 247.393,A -85,B 0,C 180,E1 -3752.344,E2 -3752.344} C_VEL
LIN {X 0,Y 545.114,Z 247.391,A -85,B 0,C 180,E1 -3754.82,E2 -3754.82} C_VEL
LIN {X 0,Y 545.039,Z 247.405,A -85,B 0,C 180,E1 -3757.242,E2 -3757.242} C_VEL
LIN {X 0,Y 545.115,Z 247.39,A -85,B 0,C 180,E1 -3760.414,E2 -3760.414} C_VEL
LIN {X 0,Y 545.069,Z 247.405,A -85,B 0,C 180,E1 -3763.521,E2 -3763.521} C_VEL
LIN {X 0,Y 545.089,Z 247.399,A -85,B 0,C 180,E1 -3765.819,E2 -3765.819} C_VEL
LIN {X 0,Y 545.112,Z 247.391,A -85,B 0,C 180,E1 -3768.849,E2 -3768.849} C_VEL
LIN {X 0,Y 545.127,Z 247.393,A -85,B 0,C 180,E1 -3771.846,E2 -3771.846} C_VEL
LIN {X 0,Y 545.2,Z 247.38,A -85,B 0,C 180,E1 -3774.822,E2 -3774.822} C_VEL
LIN {X 0,Y 545.189,Z 247.387,A -85,B 0,C 180,E1 -3777.783,E2 -3777.783} C_VEL
LIN {X 0,Y 545.208,Z 247.379,A -85,B 0,C 180,E1 -3780.738,E2 -3780.738} C_VEL
LIN {X 0,Y 545.169,Z 247.385,A -85,B 0,C 180,E1 -3782.955,E2 -3782.955} C_VEL
LIN {X 0,Y 545.163,Z 247.388,A -85,B 0,C 180,E1 -3785.919,E2 -3785.919} C_VEL
LIN {X 0,Y 545.115,Z 247.391,A -85,B 0,C 180,E1 -3788.899,E2 -3788.899} C_VEL
LIN {X 0,Y 545.127,Z 247.393,A -85,B 0,C 180,E1 -3791.904,E2 -3791.904} C_VEL
LIN {X 0,Y 545.077,Z 247.396,A -85,B 0,C 180,E1 -3794.943,E2 -3794.943} C_VEL
LIN {X 0,Y 545.075,Z 247.398,A -85,B 0,C 180,E1 -3798.025,E2 -3798.025} C_VEL
LIN {X 0,Y 545.09,Z 247.394,A -85,B 0,C 180,E1 -3800.371,E2 -3800.371} C_VEL
LIN {X 0,Y 545.082,Z 247.404,A -85,B 0,C 180,E1 -3803.558,E2 -3803.558} C_VEL
LIN {X 0,Y 545.08,Z 247.398,A -85,B 0,C 180,E1 -3806,E2 -3806} C_VEL
LIN {X 0,Y 545.081,Z 247.395,A -85,B 0,C 180,E1 -3808.748,E2 -3808.748} C_VEL
LIN {X 0,Y 545.069,Z 247.404,A -85,B 0,C 180,E1 -3811.682,E2 -3811.682} C_VEL
LIN {X 0,Y 545.076,Z 247.395,A -85,B 0,C 180,E1 -3814.562,E2 -3814.562} C_VEL
LIN {X 0,Y 545.055,Z 247.4,A -85,B 0,C 180,E1 -3817.017,E2 -3817.017} C_VEL
LIN {X 0,Y 544.35,Z 247.494,A -85,B 0,C 180,E1 -3817.633,E2 -3817.633} C_VEL
LIN {X 0,Y 541.497,Z 247.85,A -85,B 0,C 180,E1 -3818.635,E2 -3818.635} C_VEL
LIN {X 0,Y 539.115,Z 248.145,A -85,B 0,C 180,E1 -3819.44,E2 -3819.44} C_VEL
LIN {X 0,Y 538.101,Z 248.267,A -85,B 0,C 180,E1 -3820.062,E2 -3820.062} C_VEL
LIN {X 0,Y 538.022,Z 248.275,A -85,B 0,C 180,E1 -3820.273,E2 -3820.273} C_VEL
LIN {X 0,Y 538.023,Z 248.276,A -85,B 0,C 180,E1 -3822.988,E2 -3822.988} C_VEL
LIN {X 0,Y 538.02,Z 248.278,A -85,B 0,C 180,E1 -3825.925,E2 -3825.925} C_VEL
LIN {X 0,Y 538.069,Z 248.273,A -85,B 0,C 180,E1 -3829.249,E2 -3829.249} C_VEL
LIN {X 0,Y 537.984,Z 248.281,A -85,B 0,C 180,E1 -3832.122,E2 -3832.122} C_VEL
LIN {X 0,Y 538.002,Z 248.278,A -85,B 0,C 180,E1 -3834.917,E2 -3834.917} C_VEL
LIN {X 0,Y 538.022,Z 248.283,A -85,B 0,C 180,E1 -3837.618,E2 -3837.618} C_VEL
LIN {X 0,Y 538.009,Z 248.277,A -85,B 0,C 180,E1 -3840.239,E2 -3840.239} C_VEL
LIN {X 0,Y 538.057,Z 248.27,A -85,B 0,C 180,E1 -3842.796,E2 -3842.796} C_VEL
LIN {X 0,Y 538.044,Z 248.277,A -85,B 0,C 180,E1 -3845.293,E2 -3845.293} C_VEL
LIN {X 0,Y 538.023,Z 248.277,A -85,B 0,C 180,E1 -3848.037,E2 -3848.037} C_VEL
LIN {X 0,Y 538.029,Z 248.274,A -85,B 0,C 180,E1 -3850.94,E2 -3850.94} C_VEL
LIN {X 0,Y 538.018,Z 248.28,A -85,B 0,C 180,E1 -3853.299,E2 -3853.299} C_VEL
LIN {X 0,Y 538.055,Z 248.279,A -85,B 0,C 180,E1 -3855.631,E2 -3855.631} C_VEL
LIN {X 0,Y 538.081,Z 248.267,A -85,B 0,C 180,E1 -3858.702,E2 -3858.702} C_VEL
LIN {X 0,Y 538.078,Z 248.274,A -85,B 0,C 180,E1 -3861.739,E2 -3861.739} C_VEL
LIN {X 0,Y 538.152,Z 248.258,A -85,B 0,C 180,E1 -3864.755,E2 -3864.755} C_VEL
LIN {X 0,Y 538.154,Z 248.264,A -85,B 0,C 180,E1 -3867.755,E2 -3867.755} C_VEL
LIN {X 0,Y 538.172,Z 248.256,A -85,B 0,C 180,E1 -3870.748,E2 -3870.748} C_VEL
LIN {X 0,Y 538.129,Z 248.262,A -85,B 0,C 180,E1 -3872.994,E2 -3872.994} C_VEL
LIN {X 0,Y 538.101,Z 248.268,A -85,B 0,C 180,E1 -3875.997,E2 -3875.997} C_VEL
LIN {X 0,Y 538.051,Z 248.272,A -85,B 0,C 180,E1 -3879.018,E2 -3879.018} C_VEL
LIN {X 0,Y 538.072,Z 248.271,A -85,B 0,C 180,E1 -3882.062,E2 -3882.062} C_VEL
LIN {X 0,Y 538.032,Z 248.276,A -85,B 0,C 180,E1 -3885.144,E2 -3885.144} C_VEL
LIN {X 0,Y 538.007,Z 248.277,A -85,B 0,C 180,E1 -3888.27,E2 -3888.27} C_VEL
LIN {X 0,Y 538.027,Z 248.274,A -85,B 0,C 180,E1 -3890.651,E2 -3890.651} C_VEL
LIN {X 0,Y 537.994,Z 248.283,A -85,B 0,C 180,E1 -3893.878,E2 -3893.878} C_VEL
LIN {X 0,Y 538.023,Z 248.274,A -85,B 0,C 180,E1 -3896.367,E2 -3896.367} C_VEL
LIN {X 0,Y 538.018,Z 248.276,A -85,B 0,C 180,E1 -3898.933,E2 -3898.933} C_VEL
LIN {X 0,Y 537.999,Z 248.284,A -85,B 0,C 180,E1 -3901.887,E2 -3901.887} C_VEL
LIN {X 0,Y 537.932,Z 248.453,A -85,B 0,C 180,E1 -3903.334,E2 -3903.334} C_VEL
LIN {X 0,Y 537.792,Z 261.681,A -85,B 0,C 180,E1 -3906.483,E2 -3906.483} C_VEL
LIN {X 0,Y 537.757,Z 265.779,A -85,B 0,C 180,E1 -3907.459,E2 -3907.459} C_VEL
LIN {X 0,Y 538.869,Z 273.291,A -85,B 0,C 180,E1 -3907.6,E2 -3907.6} C_VEL
LIN {X 0,Y 538.611,Z 340.909,A -85,B 0,C 180,E1 -3908.522,E2 -3908.522} C_VEL
LIN {X 0,Y 538.488,Z 350.871,A -85,B 0,C 180,E1 -3908.763,E2 -3908.763} C_VEL
LIN {X 0,Y 538.407,Z 361.661,A -85,B 0,C 180,E1 -3909.156,E2 -3909.156} C_VEL
LIN {X 0,Y 538.275,Z 371.505,A -85,B 0,C 180,E1 -3909.661,E2 -3909.661} C_VEL
LIN {X 0,Y 538.161,Z 380.63,A -85,B 0,C 180,E1 -3910.272,E2 -3910.272} C_VEL
LIN {X 0,Y 538.014,Z 388.248,A -85,B 0,C 180,E1 -3910.901,E2 -3910.901} C_VEL
LIN {X 0,Y 537.898,Z 394.617,A -85,B 0,C 180,E1 -3911.534,E2 -3911.534} C_VEL
LIN {X 0,Y 537.793,Z 401.05,A -85,B 0,C 180,E1 -3912.305,E2 -3912.305} C_VEL
LIN {X 0,Y 537.731,Z 406.728,A -85,B 0,C 180,E1 -3913.133,E2 -3913.133} C_VEL
LIN {X 0,Y 537.633,Z 411.734,A -85,B 0,C 180,E1 -3914.032,E2 -3914.032} C_VEL
LIN {X 0,Y 537.591,Z 415.6,A -85,B 0,C 180,E1 -3914.905,E2 -3914.905} C_VEL
LIN {X 0,Y 537.552,Z 419.707,A -85,B 0,C 180,E1 -3916.139,E2 -3916.139} C_VEL
LIN {X 0,Y 537.494,Z 421.912,A -85,B 0,C 180,E1 -3917.164,E2 -3917.164} C_VEL
LIN {X 0,Y 537.486,Z 423.138,A -85,B 0,C 180,E1 -3918.184,E2 -3918.184} C_VEL
LIN {X 0,Y 537.476,Z 423.389,A -85,B 0,C 180,E1 -3919.322,E2 -3919.322} C_VEL
LIN {X 0,Y 537.446,Z 422.491,A -85,B 0,C 180,E1 -3920.489,E2 -3920.489} C_VEL
LIN {X 0,Y 537.528,Z 420.374,A -85,B 0,C 180,E1 -3921.671,E2 -3921.671} C_VEL
LIN {X 0,Y 537.593,Z 416.817,A -85,B 0,C 180,E1 -3922.886,E2 -3922.886} C_VEL
LIN {X 0,Y 537.673,Z 412.194,A -85,B 0,C 180,E1 -3923.972,E2 -3923.972} C_VEL
LIN {X 0,Y 537.728,Z 407.14,A -85,B 0,C 180,E1 -3924.897,E2 -3924.897} C_VEL
LIN {X 0,Y 537.798,Z 402.374,A -85,B 0,C 180,E1 -3925.614,E2 -3925.614} C_VEL
LIN {X 0,Y 537.876,Z 396.227,A -85,B 0,C 180,E1 -3926.381,E2 -3926.381} C_VEL
LIN {X 0,Y 538.026,Z 389.614,A -85,B 0,C 180,E1 -3927.065,E2 -3927.065} C_VEL
LIN {X 0,Y 538.143,Z 383.157,A -85,B 0,C 180,E1 -3927.627,E2 -3927.627} C_VEL
LIN {X 0,Y 538.285,Z 375.118,A -85,B 0,C 180,E1 -3928.203,E2 -3928.203} C_VEL
LIN {X 0,Y 538.347,Z 366.744,A -85,B 0,C 180,E1 -3928.686,E2 -3928.686} C_VEL
LIN {X 0,Y 538.435,Z 358.151,A -85,B 0,C 180,E1 -3929.074,E2 -3929.074} C_VEL
LIN {X 0,Y 538.562,Z 348.969,A -85,B 0,C 180,E1 -3929.381,E2 -3929.381} C_VEL
LIN {X 0,Y 538.634,Z 339.768,A -85,B 0,C 180,E1 -3929.589,E2 -3929.589} C_VEL
LIN {X 0,Y 538.819,Z 272.289,A -85,B 0,C 180,E1 -3930.504,E2 -3930.504} C_VEL
LIN {X 0,Y 537.797,Z 265.593,A -85,B 0,C 180,E1 -3930.63,E2 -3930.63} C_VEL
LIN {X 0,Y 537.806,Z 252.638,A -85,B 0,C 180,E1 -3933.413,E2 -3933.413} C_VEL
LIN {X 0,Y 537.831,Z 248.307,A -85,B 0,C 180,E1 -3934.349,E2 -3934.349} C_VEL
LIN {X 0,Y 537.994,Z 248.283,A -85,B 0,C 180,E1 -3936.122,E2 -3936.122} C_VEL
LIN {X 0,Y 538.031,Z 248.276,A -85,B 0,C 180,E1 -3939.349,E2 -3939.349} C_VEL
LIN {X 0,Y 538.061,Z 248.279,A -85,B 0,C 180,E1 -3942.518,E2 -3942.518} C_VEL
LIN {X 0,Y 538.053,Z 248.271,A -85,B 0,C 180,E1 -3945.631,E2 -3945.631} C_VEL
LIN {X 0,Y 538.079,Z 248.274,A -85,B 0,C 180,E1 -3948.702,E2 -3948.702} C_VEL
LIN {X 0,Y 538.081,Z 248.268,A -85,B 0,C 180,E1 -3951.74,E2 -3951.74} C_VEL
LIN {X 0,Y 538.175,Z 248.26,A -85,B 0,C 180,E1 -3954.756,E2 -3954.756} C_VEL
LIN {X 0,Y 538.158,Z 248.257,A -85,B 0,C 180,E1 -3957.755,E2 -3957.755} C_VEL
LIN {X 0,Y 538.177,Z 248.259,A -85,B 0,C 180,E1 -3960.749,E2 -3960.749} C_VEL
LIN {X 0,Y 538.134,Z 248.262,A -85,B 0,C 180,E1 -3962.995,E2 -3962.995} C_VEL
LIN {X 0,Y 538.116,Z 248.264,A -85,B 0,C 180,E1 -3965.998,E2 -3965.998} C_VEL
LIN {X 0,Y 538.068,Z 248.27,A -85,B 0,C 180,E1 -3969.018,E2 -3969.018} C_VEL
LIN {X 0,Y 538.074,Z 248.27,A -85,B 0,C 180,E1 -3972.063,E2 -3972.063} C_VEL
LIN {X 0,Y 538.037,Z 248.273,A -85,B 0,C 180,E1 -3975.144,E2 -3975.144} C_VEL
LIN {X 0,Y 538.027,Z 248.278,A -85,B 0,C 180,E1 -3978.271,E2 -3978.271} C_VEL
LIN {X 0,Y 538.035,Z 248.277,A -85,B 0,C 180,E1 -3980.652,E2 -3980.652} C_VEL
LIN {X 0,Y 538.017,Z 248.276,A -85,B 0,C 180,E1 -3983.888,E2 -3983.888} C_VEL
LIN {X 0,Y 538.044,Z 248.277,A -85,B 0,C 180,E1 -3986.367,E2 -3986.367} C_VEL
LIN {X 0,Y 538.05,Z 248.271,A -85,B 0,C 180,E1 -3988.939,E2 -3988.939} C_VEL
LIN {X 0,Y 538.008,Z 248.277,A -85,B 0,C 180,E1 -3991.889,E2 -3991.889} C_VEL
LIN {X 0,Y 538.025,Z 248.281,A -85,B 0,C 180,E1 -3994.622,E2 -3994.622} C_VEL
LIN {X 0,Y 538.004,Z 248.276,A -85,B 0,C 180,E1 -3997.172,E2 -3997.172} C_VEL
LIN {X 0,Y 538.049,Z 248.272,A -85,B 0,C 180,E1 -3999.795,E2 -3999.795} C_VEL
LIN {X 0,Y 538.014,Z 248.279,A -85,B 0,C 180,E1 -4002.787,E2 -4002.787} C_VEL
LIN {X 0,Y 538.02,Z 248.276,A -85,B 0,C 180,E1 -4005.927,E2 -4005.927} C_VEL
LIN {X 0,Y 538.045,Z 248.272,A -85,B 0,C 180,E1 -4009.225,E2 -4009.225} C_VEL
LIN {X 0,Y 537.989,Z 248.282,A -85,B 0,C 180,E1 -4012.123,E2 -4012.123} C_VEL
LIN {X 0,Y 538.009,Z 248.279,A -85,B 0,C 180,E1 -4014.917,E2 -4014.917} C_VEL
LIN {X 0,Y 538.024,Z 248.274,A -85,B 0,C 180,E1 -4017.619,E2 -4017.619} C_VEL
LIN {X 0,Y 538.012,Z 248.282,A -85,B 0,C 180,E1 -4020.239,E2 -4020.239} C_VEL
LIN {X 0,Y 538.047,Z 248.277,A -85,B 0,C 180,E1 -4022.796,E2 -4022.796} C_VEL
LIN {X 0,Y 538.022,Z 248.277,A -85,B 0,C 180,E1 -4025.292,E2 -4025.292} C_VEL
LIN {X 0,Y 538.038,Z 248.367,A -85,B 0,C 180,E1 -4026.752,E2 -4026.752} C_VEL
LIN {X 0,Y 538.728,Z 253.31,A -85,B 0,C 180,E1 -4027.569,E2 -4027.569} C_VEL
LIN {X 0,Y 538.537,Z 268.495,A -85,B 0,C 180,E1 -4029.987,E2 -4029.987} C_VEL
LIN {X 0,Y 538.334,Z 285.654,A -85,B 0,C 180,E1 -4032.723,E2 -4032.723} C_VEL
LIN {X 0,Y 538.12,Z 303.943,A -85,B 0,C 180,E1 -4035.633,E2 -4035.633} C_VEL
LIN {X 0,Y 537.934,Z 321.484,A -85,B 0,C 180,E1 -4038.4,E2 -4038.4} C_VEL
LIN {X 0,Y 538.839,Z 331.488,A -85,B 0,C 180,E1 -4038.553,E2 -4038.553} C_VEL
LIN {X 0,Y 538.628,Z 399.402,A -85,B 0,C 180,E1 -4039.475,E2 -4039.475} C_VEL
LIN {X 0,Y 538.502,Z 409.189,A -85,B 0,C 180,E1 -4039.71,E2 -4039.71} C_VEL
LIN {X 0,Y 538.352,Z 420.856,A -85,B 0,C 180,E1 -4040.135,E2 -4040.135} C_VEL
LIN {X 0,Y 538.214,Z 431.567,A -85,B 0,C 180,E1 -4040.701,E2 -4040.701} C_VEL
LIN {X 0,Y 538.102,Z 439.947,A -85,B 0,C 180,E1 -4041.267,E2 -4041.267} C_VEL
LIN {X 0,Y 537.959,Z 447.875,A -85,B 0,C 180,E1 -4041.927,E2 -4041.927} C_VEL
LIN {X 0,Y 537.851,Z 455.288,A -85,B 0,C 180,E1 -4042.681,E2 -4042.681} C_VEL
LIN {X 0,Y 537.773,Z 462.194,A -85,B 0,C 180,E1 -4043.54,E2 -4043.54} C_VEL
LIN {X 0,Y 537.651,Z 468.717,A -85,B 0,C 180,E1 -4044.562,E2 -4044.562} C_VEL
LIN {X 0,Y 537.602,Z 473.365,A -85,B 0,C 180,E1 -4045.502,E2 -4045.502} C_VEL
LIN {X 0,Y 537.599,Z 476.386,A -85,B 0,C 180,E1 -4046.252,E2 -4046.252} C_VEL
LIN {X 0,Y 537.562,Z 478.726,A -85,B 0,C 180,E1 -4047.003,E2 -4047.003} C_VEL
LIN {X 0,Y 537.491,Z 480.484,A -85,B 0,C 180,E1 -4047.752,E2 -4047.752} C_VEL
LIN {X 0,Y 537.45,Z 481.745,A -85,B 0,C 180,E1 -4048.502,E2 -4048.502} C_VEL
LIN {X 0,Y 537.44,Z 482.531,A -85,B 0,C 180,E1 -4049.251,E2 -4049.251} C_VEL
LIN {X 0,Y 537.441,Z 482.829,A -85,B 0,C 180,E1 -4050,E2 -4050} C_VEL
LIN {X 0,Y 537.44,Z 482.531,A -85,B 0,C 180,E1 -4050.749,E2 -4050.749} C_VEL
LIN {X 0,Y 537.45,Z 481.746,A -85,B 0,C 180,E1 -4051.499,E2 -4051.499} C_VEL
LIN {X 0,Y 537.491,Z 480.486,A -85,B 0,C 180,E1 -4052.248,E2 -4052.248} C_VEL
LIN {X 0,Y 537.588,Z 477.569,A -85,B 0,C 180,E1 -4053.373,E2 -4053.373} C_VEL
LIN {X 0,Y 537.625,Z 474.906,A -85,B 0,C 180,E1 -4054.123,E2 -4054.123} C_VEL
LIN {X 0,Y 537.604,Z 469.689,A -85,B 0,C 180,E1 -4055.251,E2 -4055.251} C_VEL
LIN {X 0,Y 537.78,Z 463.859,A -85,B 0,C 180,E1 -4056.226,E2 -4056.226} C_VEL
LIN {X 0,Y 537.853,Z 457.026,A -85,B 0,C 180,E1 -4057.131,E2 -4057.131} C_VEL
LIN {X 0,Y 537.936,Z 448.94,A -85,B 0,C 180,E1 -4057.979,E2 -4057.979} C_VEL
LIN {X 0,Y 538.097,Z 441.226,A -85,B 0,C 180,E1 -4058.638,E2 -4058.638} C_VEL
LIN {X 0,Y 538.207,Z 433.122,A -85,B 0,C 180,E1 -4059.205,E2 -4059.205} C_VEL
LIN {X 0,Y 538.324,Z 424.725,A -85,B 0,C 180,E1 -4059.677,E2 -4059.677} C_VEL
LIN {X 0,Y 538.439,Z 416.15,A -85,B 0,C 180,E1 -4060.054,E2 -4060.054} C_VEL
LIN {X 0,Y 538.539,Z 406.754,A -85,B 0,C 180,E1 -4060.361,E2 -4060.361} C_VEL
LIN {X 0,Y 538.682,Z 395.587,A -85,B 0,C 180,E1 -4060.596,E2 -4060.596} C_VEL
LIN {X 0,Y 538.703,Z 328.197,A -85,B 0,C 180,E1 -4061.494,E2 -4061.494} C_VEL
LIN {X 0,Y 537.955,Z 321.605,A -85,B 0,C 180,E1 -4061.617,E2 -4061.617} C_VEL
LIN {X 0,Y 538.227,Z 304.384,A -85,B 0,C 180,E1 -4064.365,E2 -4064.365} C_VEL
LIN {X 0,Y 538.416,Z 285.077,A -85,B 0,C 180,E1 -4067.471,E2 -4067.471} C_VEL
LIN {X 0,Y 538.712,Z 267.788,A -85,B 0,C 180,E1 -4070.281,E2 -4070.281} C_VEL
LIN {X 0,Y 538.952,Z 253.6,A -85,B 0,C 180,E1 -4072.624,E2 -4072.624} C_VEL
LIN {X 0,Y 538.057,Z 248.279,A -85,B 0,C 180,E1 -4073.576,E2 -4073.576} C_VEL
LIN {X 0,Y 538.037,Z 248.273,A -85,B 0,C 180,E1 -4076.367,E2 -4076.367} C_VEL
LIN {X 0,Y 538.03,Z 248.275,A -85,B 0,C 180,E1 -4078.933,E2 -4078.933} C_VEL
LIN {X 0,Y 538.01,Z 248.279,A -85,B 0,C 180,E1 -4081.887,E2 -4081.887} C_VEL
LIN {X 0,Y 538.016,Z 248.274,A -85,B 0,C 180,E1 -4084.618,E2 -4084.618} C_VEL
LIN {X 0,Y 538.004,Z 248.28,A -85,B 0,C 180,E1 -4087.17,E2 -4087.17} C_VEL
LIN {X 0,Y 538.02,Z 248.279,A -85,B 0,C 180,E1 -4089.796,E2 -4089.796} C_VEL
LIN {X 0,Y 538.017,Z 248.275,A -85,B 0,C 180,E1 -4092.785,E2 -4092.785} C_VEL
LIN {X 0,Y 538.019,Z 248.278,A -85,B 0,C 180,E1 -4095.926,E2 -4095.926} C_VEL
LIN {X 0,Y 538.052,Z 248.275,A -85,B 0,C 180,E1 -4099.251,E2 -4099.251} C_VEL
LIN {X 0,Y 537.99,Z 248.279,A -85,B 0,C 180,E1 -4102.122,E2 -4102.122} C_VEL
LIN {X 0,Y 538.008,Z 248.277,A -85,B 0,C 180,E1 -4104.916,E2 -4104.916} C_VEL
LIN {X 0,Y 538.015,Z 248.283,A -85,B 0,C 180,E1 -4107.617,E2 -4107.617} C_VEL
LIN {X 0,Y 538.013,Z 248.276,A -85,B 0,C 180,E1 -4110.238,E2 -4110.238} C_VEL
LIN {X 0,Y 538.067,Z 248.269,A -85,B 0,C 180,E1 -4112.796,E2 -4112.796} C_VEL
LIN {X 0,Y 538.046,Z 248.276,A -85,B 0,C 180,E1 -4115.292,E2 -4115.292} C_VEL
LIN {X 0,Y 538.01,Z 248.278,A -85,B 0,C 180,E1 -4118.041,E2 -4118.041} C_VEL
LIN {X 0,Y 538.032,Z 248.274,A -85,B 0,C 180,E1 -4120.939,E2 -4120.939} C_VEL
LIN {X 0,Y 538.02,Z 248.28,A -85,B 0,C 180,E1 -4123.298,E2 -4123.298} C_VEL
LIN {X 0,Y 538.058,Z 248.278,A -85,B 0,C 180,E1 -4125.63,E2 -4125.63} C_VEL
LIN {X 0,Y 538.071,Z 248.268,A -85,B 0,C 180,E1 -4128.701,E2 -4128.701} C_VEL
LIN {X 0,Y 538.084,Z 248.272,A -85,B 0,C 180,E1 -4131.739,E2 -4131.739} C_VEL
LIN {X 0,Y 538.157,Z 248.257,A -85,B 0,C 180,E1 -4134.754,E2 -4134.754} C_VEL
LIN {X 0,Y 538.161,Z 248.263,A -85,B 0,C 180,E1 -4137.754,E2 -4137.754} C_VEL
LIN {X 0,Y 538.178,Z 248.255,A -85,B 0,C 180,E1 -4140.748,E2 -4140.748} C_VEL
LIN {X 0,Y 538.136,Z 248.262,A -85,B 0,C 180,E1 -4142.994,E2 -4142.994} C_VEL
LIN {X 0,Y 538.116,Z 248.265,A -85,B 0,C 180,E1 -4145.997,E2 -4145.997} C_VEL
LIN {X 0,Y 538.065,Z 248.271,A -85,B 0,C 180,E1 -4149.017,E2 -4149.017} C_VEL
LIN {X 0,Y 538.075,Z 248.269,A -85,B 0,C 180,E1 -4152.062,E2 -4152.062} C_VEL
LIN {X 0,Y 538.037,Z 248.275,A -85,B 0,C 180,E1 -4155.143,E2 -4155.143} C_VEL
LIN {X 0,Y 538.027,Z 248.274,A -85,B 0,C 180,E1 -4158.269,E2 -4158.269} C_VEL
LIN {X 0,Y 538.034,Z 248.272,A -85,B 0,C 180,E1 -4160.651,E2 -4160.651} C_VEL
LIN {X 0,Y 538.015,Z 248.279,A -85,B 0,C 180,E1 -4163.887,E2 -4163.887} C_VEL
LIN {X 0,Y 538.041,Z 248.272,A -85,B 0,C 180,E1 -4166.366,E2 -4166.366} C_VEL
LIN {X 0,Y 538.023,Z 248.275,A -85,B 0,C 180,E1 -4168.933,E2 -4168.933} C_VEL
LIN {X 0,Y 538.018,Z 248.279,A -85,B 0,C 180,E1 -4171.89,E2 -4171.89} C_VEL
LIN {X 0,Y 538.026,Z 248.273,A -85,B 0,C 180,E1 -4174.621,E2 -4174.621} C_VEL
LIN {X 0,Y 537.998,Z 248.281,A -85,B 0,C 180,E1 -4177.17,E2 -4177.17} C_VEL
LIN {X 0,Y 538.022,Z 248.275,A -85,B 0,C 180,E1 -4180.273,E2 -4180.273} C_VEL
LIN {X 0,Y 537.363,Z 248.358,A -85,B 0,C 180,E1 -4180.898,E2 -4180.898} C_VEL
LIN {X 0,Y 534.509,Z 248.72,A -85,B 0,C 180,E1 -4181.913,E2 -4181.913} C_VEL
LIN {X 0,Y 532.087,Z 249.026,A -85,B 0,C 180,E1 -4182.73,E2 -4182.73} C_VEL
LIN {X 0,Y 531.041,Z 249.153,A -85,B 0,C 180,E1 -4183.361,E2 -4183.361} C_VEL
LIN {X 0,Y 530.953,Z 249.161,A -85,B 0,C 180,E1 -4183.575,E2 -4183.575} C_VEL
LIN {X 0,Y 530.957,Z 249.154,A -85,B 0,C 180,E1 -4186.505,E2 -4186.505} C_VEL
LIN {X 0,Y 531.017,Z 249.156,A -85,B 0,C 180,E1 -4189.571,E2 -4189.571} C_VEL
LIN {X 0,Y 530.96,Z 249.154,A -85,B 0,C 180,E1 -4192.576,E2 -4192.576} C_VEL
LIN {X 0,Y 530.987,Z 249.156,A -85,B 0,C 180,E1 -4195.311,E2 -4195.311} C_VEL
LIN {X 0,Y 530.973,Z 249.155,A -85,B 0,C 180,E1 -4198.033,E2 -4198.033} C_VEL
LIN {X 0,Y 530.98,Z 249.152,A -85,B 0,C 180,E1 -4200.874,E2 -4200.874} C_VEL
LIN {X 0,Y 530.997,Z 249.154,A -85,B 0,C 180,E1 -4203.256,E2 -4203.256} C_VEL
LIN {X 0,Y 530.999,Z 249.153,A -85,B 0,C 180,E1 -4205.955,E2 -4205.955} C_VEL
LIN {X 0,Y 530.996,Z 249.152,A -85,B 0,C 180,E1 -4209.062,E2 -4209.062} C_VEL
LIN {X 0,Y 531.007,Z 249.149,A -85,B 0,C 180,E1 -4212.278,E2 -4212.278} C_VEL
LIN {X 0,Y 531.01,Z 249.154,A -85,B 0,C 180,E1 -4215.436,E2 -4215.436} C_VEL
LIN {X 0,Y 531.038,Z 249.144,A -85,B 0,C 180,E1 -4218.55,E2 -4218.55} C_VEL
LIN {X 0,Y 531.047,Z 249.152,A -85,B 0,C 180,E1 -4221.629,E2 -4221.629} C_VEL
LIN {X 0,Y 531.11,Z 249.135,A -85,B 0,C 180,E1 -4224.685,E2 -4224.685} C_VEL
LIN {X 0,Y 531.127,Z 249.14,A -85,B 0,C 180,E1 -4227.725,E2 -4227.725} C_VEL
LIN {X 0,Y 531.142,Z 249.131,A -85,B 0,C 180,E1 -4230.758,E2 -4230.758} C_VEL
LIN {X 0,Y 531.096,Z 249.139,A -85,B 0,C 180,E1 -4233.034,E2 -4233.034} C_VEL
LIN {X 0,Y 531.057,Z 249.144,A -85,B 0,C 180,E1 -4236.077,E2 -4236.077} C_VEL
LIN {X 0,Y 531.04,Z 249.144,A -85,B 0,C 180,E1 -4238.37,E2 -4238.37} C_VEL
LIN {X 0,Y 531.056,Z 249.15,A -85,B 0,C 180,E1 -4241.679,E2 -4241.679} C_VEL
LIN {X 0,Y 531.018,Z 249.148,A -85,B 0,C 180,E1 -4244.955,E2 -4244.955} C_VEL
LIN {X 0,Y 531.005,Z 249.156,A -85,B 0,C 180,E1 -4247.722,E2 -4247.722} C_VEL
LIN {X 0,Y 531.013,Z 249.149,A -85,B 0,C 180,E1 -4250.127,E2 -4250.127} C_VEL
LIN {X 0,Y 530.932,Z 249.157,A -85,B 0,C 180,E1 -4252.573,E2 -4252.573} C_VEL
LIN {X 0,Y 530.961,Z 249.156,A -85,B 0,C 180,E1 -4255.059,E2 -4255.059} C_VEL
LIN {X 0,Y 530.997,Z 249.158,A -85,B 0,C 180,E1 -4257.596,E2 -4257.596} C_VEL
LIN {X 0,Y 530.962,Z 249.154,A -85,B 0,C 180,E1 -4260.645,E2 -4260.645} C_VEL
LIN {X 0,Y 530.879,Z 249.172,A -85,B 0,C 180,E1 -4263.292,E2 -4263.292} C_VEL
LIN {X 0,Y 530.754,Z 261.046,A -85,B 0,C 180,E1 -4266.127,E2 -4266.127} C_VEL
LIN {X 0,Y 530.747,Z 266.055,A -85,B 0,C 180,E1 -4267.311,E2 -4267.311} C_VEL
LIN {X 0,Y 531.92,Z 275.299,A -85,B 0,C 180,E1 -4267.472,E2 -4267.472} C_VEL
LIN {X 0,Y 531.642,Z 340.981,A -85,B 0,C 180,E1 -4268.381,E2 -4268.381} C_VEL
LIN {X 0,Y 531.515,Z 350.388,A -85,B 0,C 180,E1 -4268.606,E2 -4268.606} C_VEL
LIN {X 0,Y 531.469,Z 359.672,A -85,B 0,C 180,E1 -4268.935,E2 -4268.935} C_VEL
LIN {X 0,Y 531.301,Z 370.756,A -85,B 0,C 180,E1 -4269.473,E2 -4269.473} C_VEL
LIN {X 0,Y 531.17,Z 380.448,A -85,B 0,C 180,E1 -4270.116,E2 -4270.116} C_VEL
LIN {X 0,Y 531.023,Z 387.818,A -85,B 0,C 180,E1 -4270.722,E2 -4270.722} C_VEL
LIN {X 0,Y 530.87,Z 395.064,A -85,B 0,C 180,E1 -4271.446,E2 -4271.446} C_VEL
LIN {X 0,Y 530.761,Z 401.888,A -85,B 0,C 180,E1 -4272.282,E2 -4272.282} C_VEL
LIN {X 0,Y 530.684,Z 407.074,A -85,B 0,C 180,E1 -4273.053,E2 -4273.053} C_VEL
LIN {X 0,Y 530.574,Z 411.941,A -85,B 0,C 180,E1 -4273.934,E2 -4273.934} C_VEL
LIN {X 0,Y 530.551,Z 414.951,A -85,B 0,C 180,E1 -4274.592,E2 -4274.592} C_VEL
LIN {X 0,Y 530.484,Z 418.812,A -85,B 0,C 180,E1 -4275.675,E2 -4275.675} C_VEL
LIN {X 0,Y 530.451,Z 421.568,A -85,B 0,C 180,E1 -4276.776,E2 -4276.776} C_VEL
LIN {X 0,Y 530.389,Z 423.276,A -85,B 0,C 180,E1 -4277.904,E2 -4277.904} C_VEL
LIN {X 0,Y 530.406,Z 423.872,A -85,B 0,C 180,E1 -4279.047,E2 -4279.047} C_VEL
LIN {X 0,Y 530.367,Z 422.89,A -85,B 0,C 180,E1 -4280.503,E2 -4280.503} C_VEL
LIN {X 0,Y 530.47,Z 420.161,A -85,B 0,C 180,E1 -4281.972,E2 -4281.972} C_VEL
LIN {X 0,Y 530.532,Z 416.87,A -85,B 0,C 180,E1 -4283.023,E2 -4283.023} C_VEL
LIN {X 0,Y 530.618,Z 412.139,A -85,B 0,C 180,E1 -4284.126,E2 -4284.126} C_VEL
LIN {X 0,Y 530.681,Z 407.189,A -85,B 0,C 180,E1 -4285.029,E2 -4285.029} C_VEL
LIN {X 0,Y 530.746,Z 402.364,A -85,B 0,C 180,E1 -4285.753,E2 -4285.753} C_VEL
LIN {X 0,Y 530.864,Z 396.278,A -85,B 0,C 180,E1 -4286.514,E2 -4286.514} C_VEL
LIN {X 0,Y 531.029,Z 389.271,A -85,B 0,C 180,E1 -4287.238,E2 -4287.238} C_VEL
LIN {X 0,Y 531.147,Z 381.901,A -85,B 0,C 180,E1 -4287.866,E2 -4287.866} C_VEL
LIN {X 0,Y 531.303,Z 374.428,A -85,B 0,C 180,E1 -4288.39,E2 -4288.39} C_VEL
LIN {X 0,Y 531.366,Z 365.523,A -85,B 0,C 180,E1 -4288.893,E2 -4288.893} C_VEL
LIN {X 0,Y 531.545,Z 354.403,A -85,B 0,C 180,E1 -4289.365,E2 -4289.365} C_VEL
LIN {X 0,Y 531.622,Z 342.666,A -85,B 0,C 180,E1 -4289.679,E2 -4289.679} C_VEL
LIN {X 0,Y 531.775,Z 309.7,A -85,B 0,C 180,E1 -4290.155,E2 -4290.155} C_VEL
LIN {X 0,Y 531.87,Z 272.892,A -85,B 0,C 180,E1 -4290.651,E2 -4290.651} C_VEL
LIN {X 0,Y 530.76,Z 265.711,A -85,B 0,C 180,E1 -4290.799,E2 -4290.799} C_VEL
LIN {X 0,Y 530.754,Z 252.163,A -85,B 0,C 180,E1 -4293.668,E2 -4293.668} C_VEL
LIN {X 0,Y 530.752,Z 249.189,A -85,B 0,C 180,E1 -4294.282,E2 -4294.282} C_VEL
LIN {X 0,Y 530.945,Z 249.165,A -85,B 0,C 180,E1 -4296.604,E2 -4296.604} C_VEL
LIN {X 0,Y 531.013,Z 249.151,A -85,B 0,C 180,E1 -4299.873,E2 -4299.873} C_VEL
LIN {X 0,Y 530.982,Z 249.154,A -85,B 0,C 180,E1 -4303.072,E2 -4303.072} C_VEL
LIN {X 0,Y 531.008,Z 249.148,A -85,B 0,C 180,E1 -4305.436,E2 -4305.436} C_VEL
LIN {X 0,Y 531.036,Z 249.154,A -85,B 0,C 180,E1 -4308.55,E2 -4308.55} C_VEL
LIN {X 0,Y 531.05,Z 249.143,A -85,B 0,C 180,E1 -4311.63,E2 -4311.63} C_VEL
LIN {X 0,Y 531.131,Z 249.139,A -85,B 0,C 180,E1 -4314.686,E2 -4314.686} C_VEL
LIN {X 0,Y 531.13,Z 249.132,A -85,B 0,C 180,E1 -4317.726,E2 -4317.726} C_VEL
LIN {X 0,Y 531.146,Z 249.135,A -85,B 0,C 180,E1 -4320.759,E2 -4320.759} C_VEL
LIN {X 0,Y 531.1,Z 249.138,A -85,B 0,C 180,E1 -4323.035,E2 -4323.035} C_VEL
LIN {X 0,Y 531.076,Z 249.142,A -85,B 0,C 180,E1 -4326.078,E2 -4326.078} C_VEL
LIN {X 0,Y 531.026,Z 249.146,A -85,B 0,C 180,E1 -4329.139,E2 -4329.139} C_VEL
LIN {X 0,Y 531.032,Z 249.149,A -85,B 0,C 180,E1 -4332.226,E2 -4332.226} C_VEL
LIN {X 0,Y 530.988,Z 249.15,A -85,B 0,C 180,E1 -4335.35,E2 -4335.35} C_VEL
LIN {X 0,Y 531.009,Z 249.147,A -85,B 0,C 180,E1 -4337.723,E2 -4337.723} C_VEL
LIN {X 0,Y 530.994,Z 249.15,A -85,B 0,C 180,E1 -4340.939,E2 -4340.939} C_VEL
LIN {X 0,Y 530.973,Z 249.157,A -85,B 0,C 180,E1 -4344.225,E2 -4344.225} C_VEL
LIN {X 0,Y 531.005,Z 249.154,A -85,B 0,C 180,E1 -4346.744,E2 -4346.744} C_VEL
LIN {X 0,Y 530.994,Z 249.147,A -85,B 0,C 180,E1 -4349.322,E2 -4349.322} C_VEL
LIN {X 0,Y 530.964,Z 249.157,A -85,B 0,C 180,E1 -4352.102,E2 -4352.102} C_VEL
LIN {X 0,Y 530.983,Z 249.155,A -85,B 0,C 180,E1 -4354.855,E2 -4354.855} C_VEL
LIN {X 0,Y 530.962,Z 249.152,A -85,B 0,C 180,E1 -4357.508,E2 -4357.508} C_VEL
LIN {X 0,Y 531.021,Z 249.154,A -85,B 0,C 180,E1 -4360.43,E2 -4360.43} C_VEL
LIN {X 0,Y 530.95,Z 249.154,A -85,B 0,C 180,E1 -4363.496,E2 -4363.496} C_VEL
LIN {X 0,Y 530.955,Z 249.162,A -85,B 0,C 180,E1 -4366.506,E2 -4366.506} C_VEL
LIN {X 0,Y 530.983,Z 249.154,A -85,B 0,C 180,E1 -4368.977,E2 -4368.977} C_VEL
LIN {X 0,Y 530.953,Z 249.155,A -85,B 0,C 180,E1 -4371.53,E2 -4371.53} C_VEL
LIN {X 0,Y 530.974,Z 249.161,A -85,B 0,C 180,E1 -4374.382,E2 -4374.382} C_VEL
LIN {X 0,Y 530.968,Z 249.155,A -85,B 0,C 180,E1 -4377.134,E2 -4377.134} C_VEL
LIN {X 0,Y 530.966,Z 249.155,A -85,B 0,C 180,E1 -4379.804,E2 -4379.804} C_VEL
LIN {X 0,Y 531.007,Z 249.158,A -85,B 0,C 180,E1 -4382.469,E2 -4382.469} C_VEL
LIN {X 0,Y 530.988,Z 249.156,A -85,B 0,C 180,E1 -4384.942,E2 -4384.942} C_VEL
LIN {X 0,Y 531.007,Z 249.186,A -85,B 0,C 180,E1 -4386.658,E2 -4386.658} C_VEL
LIN {X 0,Y 531.724,Z 255.433,A -85,B 0,C 180,E1 -4387.701,E2 -4387.701} C_VEL
LIN {X 0,Y 531.492,Z 270.264,A -85,B 0,C 180,E1 -4390.094,E2 -4390.094} C_VEL
LIN {X 0,Y 531.295,Z 287.605,A -85,B 0,C 180,E1 -4392.884,E2 -4392.884} C_VEL
LIN {X 0,Y 531.059,Z 307.103,A -85,B 0,C 180,E1 -4396.024,E2 -4396.024} C_VEL
LIN {X 0,Y 530.889,Z 320.982,A -85,B 0,C 180,E1 -4398.232,E2 -4398.232} C_VEL
LIN {X 0,Y 531.867,Z 331.922,A -85,B 0,C 180,E1 -4398.415,E2 -4398.415} C_VEL
LIN {X 0,Y 531.65,Z 398.749,A -85,B 0,C 180,E1 -4399.335,E2 -4399.335} C_VEL
LIN {X 0,Y 531.524,Z 408.616,A -85,B 0,C 180,E1 -4399.573,E2 -4399.573} C_VEL
LIN {X 0,Y 531.339,Z 420.339,A -85,B 0,C 180,E1 -4400.003,E2 -4400.003} C_VEL
LIN {X 0,Y 531.168,Z 431.08,A -85,B 0,C 180,E1 -4400.577,E2 -4400.577} C_VEL
LIN {X 0,Y 531.054,Z 439.476,A -85,B 0,C 180,E1 -4401.15,E2 -4401.15} C_VEL
LIN {X 0,Y 530.908,Z 447.417,A -85,B 0,C 180,E1 -4401.819,E2 -4401.819} C_VEL
LIN {X 0,Y 530.784,Z 454.842,A -85,B 0,C 180,E1 -4402.583,E2 -4402.583} C_VEL
LIN {X 0,Y 530.676,Z 462.565,A -85,B 0,C 180,E1 -4403.562,E2 -4403.562} C_VEL
LIN {X 0,Y 530.542,Z 469.262,A -85,B 0,C 180,E1 -4404.68,E2 -4404.68} C_VEL
LIN {X 0,Y 530.547,Z 474.487,A -85,B 0,C 180,E1 -4405.822,E2 -4405.822} C_VEL
LIN {X 0,Y 530.495,Z 477.158,A -85,B 0,C 180,E1 -4406.582,E2 -4406.582} C_VEL
LIN {X 0,Y 530.412,Z 480.084,A -85,B 0,C 180,E1 -4407.722,E2 -4407.722} C_VEL
LIN {X 0,Y 530.36,Z 481.349,A -85,B 0,C 180,E1 -4408.482,E2 -4408.482} C_VEL
LIN {X 0,Y 530.35,Z 482.138,A -85,B 0,C 180,E1 -4409.241,E2 -4409.241} C_VEL
LIN {X 0,Y 530.352,Z 482.438,A -85,B 0,C 180,E1 -4410,E2 -4410} C_VEL
LIN {X 0,Y 530.35,Z 482.141,A -85,B 0,C 180,E1 -4410.759,E2 -4410.759} C_VEL
LIN {X 0,Y 530.36,Z 481.356,A -85,B 0,C 180,E1 -4411.519,E2 -4411.519} C_VEL
LIN {X 0,Y 530.412,Z 480.096,A -85,B 0,C 180,E1 -4412.278,E2 -4412.278} C_VEL
LIN {X 0,Y 530.495,Z 477.176,A -85,B 0,C 180,E1 -4413.418,E2 -4413.418} C_VEL
LIN {X 0,Y 530.547,Z 474.511,A -85,B 0,C 180,E1 -4414.178,E2 -4414.178} C_VEL
LIN {X 0,Y 530.542,Z 469.291,A -85,B 0,C 180,E1 -4415.321,E2 -4415.321} C_VEL
LIN {X 0,Y 530.669,Z 462.656,A -85,B 0,C 180,E1 -4416.43,E2 -4416.43} C_VEL
LIN {X 0,Y 530.784,Z 454.899,A -85,B 0,C 180,E1 -4417.417,E2 -4417.417} C_VEL
LIN {X 0,Y 530.908,Z 447.489,A -85,B 0,C 180,E1 -4418.181,E2 -4418.181} C_VEL
LIN {X 0,Y 531.056,Z 439.554,A -85,B 0,C 180,E1 -4418.85,E2 -4418.85} C_VEL
LIN {X 0,Y 531.168,Z 431.166,A -85,B 0,C 180,E1 -4419.424,E2 -4419.424} C_VEL
LIN {X 0,Y 531.34,Z 420.443,A -85,B 0,C 180,E1 -4419.997,E2 -4419.997} C_VEL
LIN {X 0,Y 531.526,Z 409.567,A -85,B 0,C 180,E1 -4420.403,E2 -4420.403} C_VEL
LIN {X 0,Y 531.64,Z 400.172,A -85,B 0,C 180,E1 -4420.641,E2 -4420.641} C_VEL
LIN {X 0,Y 531.796,Z 366.625,A -85,B 0,C 180,E1 -4421.12,E2 -4421.12} C_VEL
LIN {X 0,Y 531.783,Z 329.081,A -85,B 0,C 180,E1 -4421.627,E2 -4421.627} C_VEL
LIN {X 0,Y 530.881,Z 321.352,A -85,B 0,C 180,E1 -4421.754,E2 -4421.754} C_VEL
LIN {X 0,Y 531.156,Z 304.04,A -85,B 0,C 180,E1 -4424.56,E2 -4424.56} C_VEL
LIN {X 0,Y 531.396,Z 285.94,A -85,B 0,C 180,E1 -4427.51,E2 -4427.51} C_VEL
LIN {X 0,Y 531.693,Z 269.599,A -85,B 0,C 180,E1 -4430.2,E2 -4430.2} C_VEL
LIN {X 0,Y 531.926,Z 254.509,A -85,B 0,C 180,E1 -4432.734,E2 -4432.734} C_VEL
LIN {X 0,Y 531,Z 249.158,A -85,B 0,C 180,E1 -4433.716,E2 -4433.716} C_VEL
LIN {X 0,Y 530.995,Z 249.151,A -85,B 0,C 180,E1 -4436.744,E2 -4436.744} C_VEL
LIN {X 0,Y 530.98,Z 249.158,A -85,B 0,C 180,E1 -4439.322,E2 -4439.322} C_VEL
LIN {X 0,Y 530.965,Z 249.154,A -85,B 0,C 180,E1 -4442.1,E2 -4442.1} C_VEL
LIN {X 0,Y 530.975,Z 249.152,A -85,B 0,C 180,E1 -4444.852,E2 -4444.852} C_VEL
LIN {X 0,Y 530.964,Z 249.162,A -85,B 0,C 180,E1 -4447.507,E2 -4447.507} C_VEL
LIN {X 0,Y 530.98,Z 249.151,A -85,B 0,C 180,E1 -4450.432,E2 -4450.432} C_VEL
LIN {X 0,Y 530.962,Z 249.159,A -85,B 0,C 180,E1 -4453.281,E2 -4453.281} C_VEL
LIN {X 0,Y 530.982,Z 249.159,A -85,B 0,C 180,E1 -4455.621,E2 -4455.621} C_VEL
LIN {X 0,Y 530.998,Z 249.149,A -85,B 0,C 180,E1 -4458.564,E2 -4458.564} C_VEL
LIN {X 0,Y 530.955,Z 249.164,A -85,B 0,C 180,E1 -4461.529,E2 -4461.529} C_VEL
LIN {X 0,Y 530.974,Z 249.152,A -85,B 0,C 180,E1 -4464.381,E2 -4464.381} C_VEL
LIN {X 0,Y 530.963,Z 249.157,A -85,B 0,C 180,E1 -4467.133,E2 -4467.133} C_VEL
LIN {X 0,Y 530.965,Z 249.158,A -85,B 0,C 180,E1 -4469.802,E2 -4469.802} C_VEL
LIN {X 0,Y 531.014,Z 249.147,A -85,B 0,C 180,E1 -4472.466,E2 -4472.466} C_VEL
LIN {X 0,Y 531.004,Z 249.15,A -85,B 0,C 180,E1 -4474.942,E2 -4474.942} C_VEL
LIN {X 0,Y 530.966,Z 249.153,A -85,B 0,C 180,E1 -4478.246,E2 -4478.246} C_VEL
LIN {X 0,Y 530.99,Z 249.15,A -85,B 0,C 180,E1 -4480.677,E2 -4480.677} C_VEL
LIN {X 0,Y 530.981,Z 249.154,A -85,B 0,C 180,E1 -4483.07,E2 -4483.07} C_VEL
LIN {X 0,Y 531.013,Z 249.154,A -85,B 0,C 180,E1 -4485.435,E2 -4485.435} C_VEL
LIN {X 0,Y 531.031,Z 249.145,A -85,B 0,C 180,E1 -4488.549,E2 -4488.549} C_VEL
LIN {X 0,Y 531.053,Z 249.15,A -85,B 0,C 180,E1 -4491.629,E2 -4491.629} C_VEL
LIN {X 0,Y 531.116,Z 249.134,A -85,B 0,C 180,E1 -4494.685,E2 -4494.685} C_VEL
LIN {X 0,Y 531.133,Z 249.139,A -85,B 0,C 180,E1 -4497.724,E2 -4497.724} C_VEL
LIN {X 0,Y 531.148,Z 249.13,A -85,B 0,C 180,E1 -4500.757,E2 -4500.757} C_VEL
LIN {X 0,Y 531.102,Z 249.138,A -85,B 0,C 180,E1 -4503.033,E2 -4503.033} C_VEL
LIN {X 0,Y 531.076,Z 249.141,A -85,B 0,C 180,E1 -4506.076,E2 -4506.076} C_VEL
LIN {X 0,Y 531.025,Z 249.149,A -85,B 0,C 180,E1 -4509.138,E2 -4509.138} C_VEL
LIN {X 0,Y 531.033,Z 249.145,A -85,B 0,C 180,E1 -4512.224,E2 -4512.224} C_VEL
LIN {X 0,Y 530.988,Z 249.156,A -85,B 0,C 180,E1 -4515.349,E2 -4515.349} C_VEL
LIN {X 0,Y 531.008,Z 249.154,A -85,B 0,C 180,E1 -4517.722,E2 -4517.722} C_VEL
LIN {X 0,Y 530.993,Z 249.151,A -85,B 0,C 180,E1 -4520.937,E2 -4520.937} C_VEL
LIN {X 0,Y 530.971,Z 249.153,A -85,B 0,C 180,E1 -4524.224,E2 -4524.224} C_VEL
LIN {X 0,Y 531.003,Z 249.149,A -85,B 0,C 180,E1 -4526.743,E2 -4526.743} C_VEL
LIN {X 0,Y 530.973,Z 249.158,A -85,B 0,C 180,E1 -4529.322,E2 -4529.322} C_VEL
LIN {X 0,Y 530.971,Z 249.154,A -85,B 0,C 180,E1 -4532.103,E2 -4532.103} C_VEL
LIN {X 0,Y 530.982,Z 249.152,A -85,B 0,C 180,E1 -4534.854,E2 -4534.854} C_VEL
LIN {X 0,Y 530.957,Z 249.162,A -85,B 0,C 180,E1 -4537.507,E2 -4537.507} C_VEL
LIN {X 0,Y 530.98,Z 249.151,A -85,B 0,C 180,E1 -4540.432,E2 -4540.432} C_VEL
LIN {X 0,Y 530.956,Z 249.162,A -85,B 0,C 180,E1 -4543.494,E2 -4543.494} C_VEL
LIN {X 0,Y 530.953,Z 249.161,A -85,B 0,C 180,E1 -4543.575,E2 -4543.575} C_VEL
LIN {X 0,Y 530.281,Z 249.241,A -85,B 0,C 180,E1 -4544.208,E2 -4544.208} C_VEL
LIN {X 0,Y 527.434,Z 249.597,A -85,B 0,C 180,E1 -4545.237,E2 -4545.237} C_VEL
LIN {X 0,Y 525.031,Z 249.895,A -85,B 0,C 180,E1 -4546.066,E2 -4546.066} C_VEL
LIN {X 0,Y 523.998,Z 250.021,A -85,B 0,C 180,E1 -4546.705,E2 -4546.705} C_VEL
LIN {X 0,Y 523.913,Z 250.033,A -85,B 0,C 180,E1 -4546.922,E2 -4546.922} C_VEL
LIN {X 0,Y 523.969,Z 250.029,A -85,B 0,C 180,E1 -4549.923,E2 -4549.923} C_VEL
LIN {X 0,Y 523.902,Z 250.034,A -85,B 0,C 180,E1 -4552.868,E2 -4552.868} C_VEL
LIN {X 0,Y 523.931,Z 250.037,A -85,B 0,C 180,E1 -4555.71,E2 -4555.71} C_VEL
LIN {X 0,Y 523.922,Z 250.031,A -85,B 0,C 180,E1 -4558.456,E2 -4558.456} C_VEL
LIN {X 0,Y 523.931,Z 250.033,A -85,B 0,C 180,E1 -4561.125,E2 -4561.125} C_VEL
LIN {X 0,Y 523.975,Z 250.027,A -85,B 0,C 180,E1 -4563.98,E2 -4563.98} C_VEL
LIN {X 0,Y 523.935,Z 250.032,A -85,B 0,C 180,E1 -4567.108,E2 -4567.108} C_VEL
LIN {X 0,Y 523.97,Z 250.029,A -85,B 0,C 180,E1 -4569.865,E2 -4569.865} C_VEL
LIN {X 0,Y 523.958,Z 250.027,A -85,B 0,C 180,E1 -4572.837,E2 -4572.837} C_VEL
LIN {X 0,Y 523.967,Z 250.029,A -85,B 0,C 180,E1 -4575.236,E2 -4575.236} C_VEL
LIN {X 0,Y 524.003,Z 250.021,A -85,B 0,C 180,E1 -4578.394,E2 -4578.394} C_VEL
LIN {X 0,Y 523.996,Z 250.029,A -85,B 0,C 180,E1 -4581.516,E2 -4581.516} C_VEL
LIN {X 0,Y 524.071,Z 250.012,A -85,B 0,C 180,E1 -4584.613,E2 -4584.613} C_VEL
LIN {X 0,Y 524.099,Z 250.016,A -85,B 0,C 180,E1 -4587.694,E2 -4587.694} C_VEL
LIN {X 0,Y 524.113,Z 250.007,A -85,B 0,C 180,E1 -4590.768,E2 -4590.768} C_VEL
LIN {X 0,Y 524.063,Z 250.016,A -85,B 0,C 180,E1 -4593.075,E2 -4593.075} C_VEL
LIN {X 0,Y 524.02,Z 250.02,A -85,B 0,C 180,E1 -4596.159,E2 -4596.159} C_VEL
LIN {X 0,Y 523.989,Z 250.022,A -85,B 0,C 180,E1 -4598.484,E2 -4598.484} C_VEL
LIN {X 0,Y 524.015,Z 250.026,A -85,B 0,C 180,E1 -4601.751,E2 -4601.751} C_VEL
LIN {X 0,Y 523.981,Z 250.026,A -85,B 0,C 180,E1 -4605.051,E2 -4605.051} C_VEL
LIN {X 0,Y 523.95,Z 250.031,A -85,B 0,C 180,E1 -4607.969,E2 -4607.969} C_VEL
LIN {X 0,Y 523.961,Z 250.026,A -85,B 0,C 180,E1 -4610.41,E2 -4610.41} C_VEL
LIN {X 0,Y 523.898,Z 250.035,A -85,B 0,C 180,E1 -4612.893,E2 -4612.893} C_VEL
LIN {X 0,Y 523.932,Z 250.033,A -85,B 0,C 180,E1 -4616.011,E2 -4616.011} C_VEL
LIN {X 0,Y 523.916,Z 250.032,A -85,B 0,C 180,E1 -4618.875,E2 -4618.875} C_VEL
LIN {X 0,Y 523.909,Z 250.041,A -85,B 0,C 180,E1 -4621.544,E2 -4621.544} C_VEL
LIN {X 0,Y 523.831,Z 250.217,A -85,B 0,C 180,E1 -4623.314,E2 -4623.314} C_VEL
LIN {X 0,Y 523.713,Z 262.277,A -85,B 0,C 180,E1 -4626.189,E2 -4626.189} C_VEL
LIN {X 0,Y 523.704,Z 266.31,A -85,B 0,C 180,E1 -4627.148,E2 -4627.148} C_VEL
LIN {X 0,Y 524.976,Z 274.714,A -85,B 0,C 180,E1 -4627.306,E2 -4627.306} C_VEL
LIN {X 0,Y 524.677,Z 341.737,A -85,B 0,C 180,E1 -4628.249,E2 -4628.249} C_VEL
LIN {X 0,Y 524.539,Z 351.973,A -85,B 0,C 180,E1 -4628.506,E2 -4628.506} C_VEL
LIN {X 0,Y 524.461,Z 362.693,A -85,B 0,C 180,E1 -4628.912,E2 -4628.912} C_VEL
LIN {X 0,Y 524.297,Z 372.316,A -85,B 0,C 180,E1 -4629.422,E2 -4629.422} C_VEL
LIN {X 0,Y 524.173,Z 381.539,A -85,B 0,C 180,E1 -4630.058,E2 -4630.058} C_VEL
LIN {X 0,Y 523.991,Z 389.272,A -85,B 0,C 180,E1 -4630.716,E2 -4630.716} C_VEL
LIN {X 0,Y 523.853,Z 395.015,A -85,B 0,C 180,E1 -4631.299,E2 -4631.299} C_VEL
LIN {X 0,Y 523.72,Z 401.878,A -85,B 0,C 180,E1 -4632.141,E2 -4632.141} C_VEL
LIN {X 0,Y 523.621,Z 407.547,A -85,B 0,C 180,E1 -4632.99,E2 -4632.99} C_VEL
LIN {X 0,Y 523.53,Z 412.375,A -85,B 0,C 180,E1 -4633.878,E2 -4633.878} C_VEL
LIN {X 0,Y 523.465,Z 415.741,A -85,B 0,C 180,E1 -4634.638,E2 -4634.638} C_VEL
LIN {X 0,Y 523.401,Z 419.448,A -85,B 0,C 180,E1 -4635.716,E2 -4635.716} C_VEL
LIN {X 0,Y 523.363,Z 422.021,A -85,B 0,C 180,E1 -4636.777,E2 -4636.777} C_VEL
LIN {X 0,Y 523.315,Z 423.577,A -85,B 0,C 180,E1 -4637.819,E2 -4637.819} C_VEL
LIN {X 0,Y 523.331,Z 424.206,A -85,B 0,C 180,E1 -4638.851,E2 -4638.851} C_VEL
LIN {X 0,Y 523.271,Z 423.918,A -85,B 0,C 180,E1 -4639.955,E2 -4639.955} C_VEL
LIN {X 0,Y 523.33,Z 422.373,A -85,B 0,C 180,E1 -4641.159,E2 -4641.159} C_VEL
LIN {X 0,Y 523.386,Z 420.925,A -85,B 0,C 180,E1 -4641.854,E2 -4641.854} C_VEL
LIN {X 0,Y 523.456,Z 418.133,A -85,B 0,C 180,E1 -4642.832,E2 -4642.832} C_VEL
LIN {X 0,Y 523.552,Z 413.298,A -85,B 0,C 180,E1 -4644.037,E2 -4644.037} C_VEL
LIN {X 0,Y 523.608,Z 408.479,A -85,B 0,C 180,E1 -4644.959,E2 -4644.959} C_VEL
LIN {X 0,Y 523.701,Z 402.63,A -85,B 0,C 180,E1 -4645.859,E2 -4645.859} C_VEL
LIN {X 0,Y 523.83,Z 396.526,A -85,B 0,C 180,E1 -4646.629,E2 -4646.629} C_VEL
LIN {X 0,Y 524.024,Z 389.817,A -85,B 0,C 180,E1 -4647.33,E2 -4647.33} C_VEL
LIN {X 0,Y 524.147,Z 382.949,A -85,B 0,C 180,E1 -4647.929,E2 -4647.929} C_VEL
LIN {X 0,Y 524.323,Z 375.242,A -85,B 0,C 180,E1 -4648.484,E2 -4648.484} C_VEL
LIN {X 0,Y 524.381,Z 366.599,A -85,B 0,C 180,E1 -4648.986,E2 -4648.986} C_VEL
LIN {X 0,Y 524.53,Z 357.461,A -85,B 0,C 180,E1 -4649.394,E2 -4649.394} C_VEL
LIN {X 0,Y 524.643,Z 345.821,A -85,B 0,C 180,E1 -4649.763,E2 -4649.763} C_VEL
LIN {X 0,Y 524.738,Z 328.524,A -85,B 0,C 180,E1 -4650.046,E2 -4650.046} C_VEL
LIN {X 0,Y 524.869,Z 273.313,A -85,B 0,C 180,E1 -4650.808,E2 -4650.808} C_VEL
LIN {X 0,Y 523.735,Z 265.969,A -85,B 0,C 180,E1 -4650.955,E2 -4650.955} C_VEL
LIN {X 0,Y 523.695,Z 252.793,A -85,B 0,C 180,E1 -4653.714,E2 -4653.714} C_VEL
LIN {X 0,Y 523.736,Z 250.063,A -85,B 0,C 180,E1 -4654.309,E2 -4654.309} C_VEL
LIN {X 0,Y 523.9,Z 250.041,A -85,B 0,C 180,E1 -4656.27,E2 -4656.27} C_VEL
LIN {X 0,Y 523.936,Z 250.037,A -85,B 0,C 180,E1 -4658.767,E2 -4658.767} C_VEL
LIN {X 0,Y 523.943,Z 250.031,A -85,B 0,C 180,E1 -4661.221,E2 -4661.221} C_VEL
LIN {X 0,Y 523.929,Z 250.031,A -85,B 0,C 180,E1 -4663.639,E2 -4663.639} C_VEL
LIN {X 0,Y 523.93,Z 250.033,A -85,B 0,C 180,E1 -4666.029,E2 -4666.029} C_VEL
LIN {X 0,Y 524.001,Z 250.029,A -85,B 0,C 180,E1 -4668.395,E2 -4668.395} C_VEL
LIN {X 0,Y 523.998,Z 250.022,A -85,B 0,C 180,E1 -4671.517,E2 -4671.517} C_VEL
LIN {X 0,Y 524.089,Z 250.017,A -85,B 0,C 180,E1 -4674.614,E2 -4674.614} C_VEL
LIN {X 0,Y 524.103,Z 250.007,A -85,B 0,C 180,E1 -4677.695,E2 -4677.695} C_VEL
LIN {X 0,Y 524.116,Z 250.01,A -85,B 0,C 180,E1 -4680.769,E2 -4680.769} C_VEL
LIN {X 0,Y 524.067,Z 250.014,A -85,B 0,C 180,E1 -4683.076,E2 -4683.076} C_VEL
LIN {X 0,Y 524.038,Z 250.02,A -85,B 0,C 180,E1 -4686.16,E2 -4686.16} C_VEL
LIN {X 0,Y 523.994,Z 250.022,A -85,B 0,C 180,E1 -4689.263,E2 -4689.263} C_VEL
LIN {X 0,Y 523.993,Z 250.021,A -85,B 0,C 180,E1 -4691.74,E2 -4691.74} C_VEL
LIN {X 0,Y 523.985,Z 250.024,A -85,B 0,C 180,E1 -4695.053,E2 -4695.053} C_VEL
LIN {X 0,Y 523.956,Z 250.027,A -85,B 0,C 180,E1 -4697.97,E2 -4697.97} C_VEL
LIN {X 0,Y 523.965,Z 250.032,A -85,B 0,C 180,E1 -4700.411,E2 -4700.411} C_VEL
LIN {X 0,Y 523.909,Z 250.035,A -85,B 0,C 180,E1 -4702.894,E2 -4702.894} C_VEL
LIN {X 0,Y 523.948,Z 250.025,A -85,B 0,C 180,E1 -4705.419,E2 -4705.419} C_VEL
LIN {X 0,Y 523.964,Z 250.028,A -85,B 0,C 180,E1 -4708,E2 -4708} C_VEL
LIN {X 0,Y 523.943,Z 250.032,A -85,B 0,C 180,E1 -4710.857,E2 -4710.857} C_VEL
LIN {X 0,Y 523.955,Z 250.024,A -85,B 0,C 180,E1 -4713.736,E2 -4713.736} C_VEL
LIN {X 0,Y 523.919,Z 250.039,A -85,B 0,C 180,E1 -4716.406,E2 -4716.406} C_VEL
LIN {X 0,Y 523.926,Z 250.032,A -85,B 0,C 180,E1 -4719.085,E2 -4719.085} C_VEL
LIN {X 0,Y 523.967,Z 250.025,A -85,B 0,C 180,E1 -4721.313,E2 -4721.313} C_VEL
LIN {X 0,Y 523.949,Z 250.034,A -85,B 0,C 180,E1 -4724.692,E2 -4724.692} C_VEL
LIN {X 0,Y 523.951,Z 250.029,A -85,B 0,C 180,E1 -4727.882,E2 -4727.882} C_VEL
LIN {X 0,Y 523.916,Z 250.035,A -85,B 0,C 180,E1 -4730.916,E2 -4730.916} C_VEL
LIN {X 0,Y 523.921,Z 250.032,A -85,B 0,C 180,E1 -4733.828,E2 -4733.828} C_VEL
LIN {X 0,Y 523.94,Z 250.036,A -85,B 0,C 180,E1 -4736.636,E2 -4736.636} C_VEL
LIN {X 0,Y 523.954,Z 250.028,A -85,B 0,C 180,E1 -4739.356,E2 -4739.356} C_VEL
LIN {X 0,Y 523.971,Z 250.033,A -85,B 0,C 180,E1 -4742.283,E2 -4742.283} C_VEL
LIN {X 0,Y 523.942,Z 250.037,A -85,B 0,C 180,E1 -4744.582,E2 -4744.582} C_VEL
LIN {X 0,Y 523.974,Z 250.196,A -85,B 0,C 180,E1 -4746.588,E2 -4746.588} C_VEL
LIN {X 0,Y 524.71,Z 255.846,A -85,B 0,C 180,E1 -4747.547,E2 -4747.547} C_VEL
LIN {X 0,Y 524.498,Z 269.68,A -85,B 0,C 180,E1 -4749.813,E2 -4749.813} C_VEL
LIN {X 0,Y 524.255,Z 288.334,A -85,B 0,C 180,E1 -4752.848,E2 -4752.848} C_VEL
LIN {X 0,Y 523.994,Z 307.874,A -85,B 0,C 180,E1 -4756.03,E2 -4756.03} C_VEL
LIN {X 0,Y 523.838,Z 320.595,A -85,B 0,C 180,E1 -4758.077,E2 -4758.077} C_VEL
LIN {X 0,Y 524.91,Z 332.102,A -85,B 0,C 180,E1 -4758.269,E2 -4758.269} C_VEL
LIN {X 0,Y 524.677,Z 398.095,A -85,B 0,C 180,E1 -4759.192,E2 -4759.192} C_VEL
LIN {X 0,Y 524.519,Z 408.04,A -85,B 0,C 180,E1 -4759.433,E2 -4759.433} C_VEL
LIN {X 0,Y 524.383,Z 418.667,A -85,B 0,C 180,E1 -4759.82,E2 -4759.82} C_VEL
